SPLINE
SPL {X  -124.054, Y  +777.532, Z    +0.000, E1   -54.436, E3 +106436.833}
SPL {X  -145.922, Y  +742.101, Z    +0.000, E1   -46.535, E3 +106455.102}
SPL {X  -155.216, Y  +715.293, Z    +0.000, E1   -34.460, E3 +106461.295}
SPL {X  -158.715, Y  +696.660, Z    +0.000, E1   -21.368, E3 +106463.622}
SPL {X  -159.838, Y  +683.473, Z    +0.000, E1    -9.532, E3 +106464.418}
SPL {X  -159.990, Y  +674.579, Z    +0.000, E1    -0.168, E3 +106464.601}
SPL {X  -159.990, Y  +672.677, Z    +0.000, E1    +3.879, E3 +106464.617}
SPL {X  -159.990, Y  +669.117, Z    +0.000, E1   +12.900, E3 +106464.699}
SPL {X  -159.990, Y  +663.639, Z    +0.000, E1   +26.675, E3 +106464.985}
SPL {X  -159.990, Y  +656.057, Z    +0.000, E1   +43.288, E3 +106465.641}
SPL {X  -159.990, Y  +647.797, Z    +0.000, E1   +54.469, E3 +106466.778}
SPL {X  -159.990, Y  +630.178, Z    +0.000, E1   +65.480, E3 +106470.462}
SPL {X  -159.990, Y  +547.268, Z    +0.000, E1   +73.735, E3 +106497.746}
SPL {X  -159.091, Y  +360.560, Z    +0.000, E1   +74.726, E3 +106584.072}
SPL {X  -156.418, Y  +343.879, Z    +0.000, E1   +74.473, E3 +106596.498}
SPL {X  -153.414, Y  +332.103, Z    +0.000, E1   +74.378, E3 +106604.173}
SPL {X  -141.909, Y  +303.617, Z    +0.000, E1   +76.515, E3 +106596.703}
ENDSPLINE

SPLINE
SPL {X  -142.567, Y  +304.895, Z    +0.000, E1   +75.566, E3 +106605.518}
ENDSPLINE

SPLINE
SPL {X  -141.999, Y  +303.790, Z    +0.000, E1   +74.633, E3 +106614.769}
SPL {X  -141.780, Y  +303.371, Z    +0.000, E1   +73.549, E3 +106624.343}
SPL {X  -140.619, Y  +301.190, Z    +0.000, E1   +72.741, E3 +106632.189}
SPL {X  -137.438, Y  +295.601, Z    +0.000, E1   +72.365, E3 +106638.278}
SPL {X  -134.156, Y  +290.328, Z    +0.000, E1   +71.962, E3 +106644.149}
SPL {X  -130.677, Y  +285.194, Z    +0.000, E1   +71.519, E3 +106649.954}
SPL {X  -127.147, Y  +280.390, Z    +0.000, E1   +71.042, E3 +106655.438}
SPL {X  -123.431, Y  +275.709, Z    +0.000, E1   +70.518, E3 +106660.761}
SPL {X  -120.392, Y  +272.131, Z    +0.000, E1   +70.053, E3 +106664.781}
SPL {X   -79.311, Y  +238.552, Z    +0.000, E1   +58.563, E3 +106760.020}
ENDSPLINE

SPLINE
SPL {X  -105.077, Y  +256.854, Z    +0.000, E1   +55.187, E3 +106947.573}
SPL {X  -133.208, Y  +288.886, Z    +0.000, E1   +52.003, E3 +106980.674}
SPL {X  -149.825, Y  +321.381, Z    +0.000, E1   +42.580, E3 +106993.827}
SPL {X  -157.376, Y  +348.695, Z    +0.000, E1   +27.651, E3 +106998.912}
SPL {X  -159.486, Y  +364.808, Z    +0.000, E1   +14.693, E3 +107000.415}
SPL {X  -159.964, Y  +374.630, Z    +0.000, E1    +5.249, E3 +107000.820}
SPL {X  -159.990, Y  +379.735, Z    +0.000, E1    -0.236, E3 +107000.878}
SPL {X  -159.990, Y  +384.648, Z    +0.000, E1   -11.739, E3 +107000.974}
SPL {X  -159.990, Y  +391.065, Z    +0.000, E1   -28.187, E3 +107001.302}
SPL {X  -159.990, Y  +399.326, Z    +0.000, E1   -44.934, E3 +107002.085}
SPL {X  -159.990, Y  +408.817, Z    +0.000, E1   -56.572, E3 +107003.458}
SPL {X  -159.990, Y  +426.617, Z    +0.000, E1   -66.230, E3 +107007.313}
SPL {X  -159.990, Y  +499.521, Z    +0.000, E1   -73.662, E3 +107030.640}
SPL {X  -159.629, Y  +687.249, Z    +0.000, E1   -74.539, E3 +107118.524}
SPL {X  -157.983, Y  +701.765, Z    +0.000, E1   -74.384, E3 +107128.756}
SPL {X  -155.520, Y  +714.054, Z    +0.000, E1   -74.151, E3 +107138.510}
SPL {X  -152.569, Y  +724.660, Z    +0.000, E1   -73.857, E3 +107147.745}
SPL {X  -149.625, Y  +733.149, Z    +0.000, E1   -73.553, E3 +107155.680}
SPL {X  -146.617, Y  +740.532, Z    +0.000, E1   -73.233, E3 +107162.957}
SPL {X  -143.394, Y  +747.457, Z    +0.000, E1   -72.883, E3 +107170.054}
SPL {X  -140.332, Y  +753.336, Z    +0.000, E1   -72.527, E3 +107176.329}
SPL {X  -137.187, Y  +758.820, Z    +0.000, E1   -72.156, E3 +107182.332}
SPL {X  -134.014, Y  +763.891, Z    +0.000, E1   -71.759, E3 +107188.017}
SPL {X  -130.657, Y  +768.834, Z    +0.000, E1   -71.330, E3 +107193.632}
SPL {X  -126.937, Y  +773.885, Z    +0.000, E1   -70.823, E3 +107199.434}
SPL {X  -122.983, Y  +778.833, Z    +0.000, E1   -70.262, E3 +107205.079}
SPL {X  -120.205, Y  +782.082, Z    +0.000, E1   -69.822, E3 +107208.747}
SPL {X   -75.772, Y  +817.409, Z    +0.000, E1   -56.226, E3 +107334.686}
ENDSPLINE

SPLINE
SPL {X  -124.054, Y  +777.532, Z    +0.000, E1   -54.436, E3 +107517.914}
SPL {X  -145.922, Y  +742.101, Z    +0.000, E1   -46.535, E3 +107536.184}
SPL {X  -155.216, Y  +715.293, Z    +0.000, E1   -34.460, E3 +107542.376}
SPL {X  -159.282, Y  +691.530, Z    +0.000, E1   -17.100, E3 +107545.071}
SPL {X  -159.981, Y  +678.202, Z    +0.000, E1    -4.129, E3 +107545.645}
SPL {X  -159.990, Y  +674.500, Z    +0.000, E1    +0.000, E3 +107545.682}
SPL {X  -159.990, Y  +672.677, Z    +0.000, E1    +3.879, E3 +107545.698}
SPL {X  -159.990, Y  +669.117, Z    +0.000, E1   +12.900, E3 +107545.781}
SPL {X  -159.990, Y  +665.253, Z    +0.000, E1   +22.908, E3 +107545.954}
SPL {X  -159.990, Y  +658.335, Z    +0.000, E1   +38.839, E3 +107546.499}
SPL {X  -159.990, Y  +645.786, Z    +0.000, E1   +56.338, E3 +107548.213}
SPL {X  -159.990, Y  +623.264, Z    +0.000, E1   +67.753, E3 +107553.139}
SPL {X  -159.990, Y  +547.268, Z    +0.000, E1   +73.735, E3 +107578.827}
SPL {X  -159.091, Y  +360.560, Z    +0.000, E1   +74.726, E3 +107665.154}
SPL {X  -156.418, Y  +343.879, Z    +0.000, E1   +74.473, E3 +107677.579}
SPL {X  -153.414, Y  +332.103, Z    +0.000, E1   +74.378, E3 +107685.254}
SPL {X  -141.909, Y  +303.617, Z    +0.000, E1   +76.515, E3 +107677.784}
ENDSPLINE

SPLINE
SPL {X  -142.567, Y  +304.895, Z    +0.000, E1   +75.566, E3 +107686.599}
ENDSPLINE

SPLINE
SPL {X  -141.999, Y  +303.790, Z    +0.000, E1   +74.633, E3 +107695.850}
SPL {X  -141.780, Y  +303.371, Z    +0.000, E1   +73.549, E3 +107705.424}
ENDSPLINE

SPLINE
SPL {X  -146.767, Y  +313.812, Z    +0.000, E1   +70.623, E3 +107723.087}
ENDSPLINE

SPLINE
SPL {X  -143.180, Y  +306.112, Z    +0.000, E1   +70.169, E3 +107731.789}
SPL {X  -139.769, Y  +299.645, Z    +0.000, E1   +69.722, E3 +107739.355}
SPL {X  -136.083, Y  +293.369, Z    +0.000, E1   +69.227, E3 +107746.896}
SPL {X  -132.274, Y  +287.498, Z    +0.000, E1   +68.678, E3 +107754.116}
SPL {X  -128.237, Y  +281.834, Z    +0.000, E1   +68.080, E3 +107761.152}
SPL {X  -124.030, Y  +276.439, Z    +0.000, E1   +67.412, E3 +107767.870}
SPL {X   -89.505, Y  +244.889, Z    +0.000, E1   +58.168, E3 +107849.622}
ENDSPLINE

SPLINE
SPL {X  -111.763, Y  +263.019, Z    +0.000, E1   +52.505, E3 +108031.034}
SPL {X  -139.943, Y  +299.958, Z    +0.000, E1   +46.517, E3 +108065.374}
SPL {X  -154.122, Y  +334.569, Z    +0.000, E1   +33.405, E3 +108077.208}
SPL {X  -159.233, Y  +361.951, Z    +0.000, E1   +15.631, E3 +108081.387}
SPL {X  -159.983, Y  +375.952, Z    +0.000, E1    +3.555, E3 +108082.153}
SPL {X  -159.990, Y  +379.545, Z    +0.000, E1    -0.045, E3 +108082.200}
SPL {X  -159.990, Y  +382.058, Z    +0.000, E1    -4.728, E3 +108082.232}
SPL {X  -159.990, Y  +387.492, Z    +0.000, E1   -16.478, E3 +108082.457}
SPL {X  -159.990, Y  +395.172, Z    +0.000, E1   -33.361, E3 +108083.084}
SPL {X  -159.990, Y  +405.626, Z    +0.000, E1   -49.217, E3 +108084.608}
SPL {X  -159.990, Y  +423.679, Z    +0.000, E1   -61.834, E3 +108088.879}
SPL {X  -159.990, Y  +491.183, Z    +0.000, E1   -70.406, E3 +108115.268}
SPL {X  -159.990, Y  +644.105, Z    +0.000, E1   -71.828, E3 +108199.837}
SPL {X  -159.990, Y  +665.410, Z    +0.000, E1   -71.813, E3 +108214.734}
SPL {X  -159.784, Y  +684.619, Z    +0.000, E1   -71.795, E3 +108228.338}
SPL {X  -158.321, Y  +699.551, Z    +0.000, E1   -71.633, E3 +108240.290}
SPL {X  -155.878, Y  +712.540, Z    +0.000, E1   -71.376, E3 +108251.853}
SPL {X  -152.746, Y  +724.097, Z    +0.000, E1   -71.019, E3 +108263.104}
SPL {X  -149.840, Y  +732.578, Z    +0.000, E1   -70.669, E3 +108271.930}
SPL {X  -147.044, Y  +739.548, Z    +0.000, E1   -70.332, E3 +108279.524}
SPL {X  -143.437, Y  +747.371, Z    +0.000, E1   -69.890, E3 +108288.388}
SPL {X  -139.209, Y  +755.353, Z    +0.000, E1   -69.333, E3 +108297.815}
SPL {X  -135.354, Y  +761.800, Z    +0.000, E1   -68.789, E3 +108305.678}
SPL {X  -131.547, Y  +767.562, Z    +0.000, E1   -68.238, E3 +108312.847}
SPL {X  -127.113, Y  +773.655, Z    +0.000, E1   -67.565, E3 +108320.504}
SPL {X  -123.626, Y  +778.056, Z    +0.000, E1   -66.969, E3 +108326.064}
SPL {X   -86.110, Y  +811.340, Z    +0.000, E1   -55.142, E3 +108443.974}
ENDSPLINE

SPLINE
SPL {X  -126.688, Y  +774.208, Z    +0.000, E1   -50.278, E3 +108604.622}
SPL {X  -150.887, Y  +729.697, Z    +0.000, E1   -37.846, E3 +108628.478}
SPL {X  -158.568, Y  +697.780, Z    +0.000, E1   -19.721, E3 +108634.807}
SPL {X  -159.967, Y  +679.234, Z    +0.000, E1    -4.684, E3 +108636.142}
SPL {X  -159.990, Y  +674.465, Z    +0.000, E1    +0.035, E3 +108636.225}
SPL {X  -159.990, Y  +672.210, Z    +0.000, E1    +4.112, E3 +108636.252}
SPL {X  -159.990, Y  +668.446, Z    +0.000, E1   +12.084, E3 +108636.377}
SPL {X  -159.990, Y  +663.424, Z    +0.000, E1   +23.273, E3 +108636.703}
SPL {X  -159.990, Y  +655.288, Z    +0.000, E1   +39.016, E3 +108637.592}
SPL {X  -159.990, Y  +641.020, Z    +0.000, E1   +55.512, E3 +108640.131}
SPL {X  -159.990, Y  +618.237, Z    +0.000, E1   +65.205, E3 +108646.657}
SPL {X  -159.990, Y  +545.807, Z    +0.000, E1   +71.095, E3 +108675.710}
SPL {X  -149.334, Y  +320.087, Z    +0.000, E1   +77.218, E3 +108741.528}
SPL {X  -149.265, Y  +319.910, Z    +0.000, E1   +76.148, E3 +108753.642}
SPL {X  -149.092, Y  +319.462, Z    +0.000, E1   +75.437, E3 +108761.517}
ENDSPLINE

SPLINE
SPL {X  -149.679, Y  +320.993, Z    +0.000, E1   +74.493, E3 +108770.411}
SPL {X  -149.823, Y  +321.377, Z    +0.000, E1   +73.518, E3 +108779.768}
ENDSPLINE

SPLINE
SPL {X  -149.061, Y  +319.382, Z    +0.000, E1   +72.547, E3 +108790.010}
SPL {X  -148.201, Y  +317.223, Z    +0.000, E1   +71.184, E3 +108803.334}
SPL {X  -144.085, Y  +307.957, Z    +0.000, E1   +70.311, E3 +108816.581}
SPL {X  -139.769, Y  +299.645, Z    +0.000, E1   +69.722, E3 +108826.312}
SPL {X  -136.083, Y  +293.369, Z    +0.000, E1   +69.227, E3 +108833.853}
SPL {X  -132.274, Y  +287.498, Z    +0.000, E1   +68.678, E3 +108841.072}
SPL {X  -128.237, Y  +281.834, Z    +0.000, E1   +68.080, E3 +108848.109}
SPL {X  -124.030, Y  +276.439, Z    +0.000, E1   +67.412, E3 +108854.826}
SPL {X   -89.505, Y  +244.889, Z    +0.000, E1   +58.168, E3 +108936.578}
ENDSPLINE

SPLINE
SPL {X  -111.763, Y  +263.019, Z    +0.000, E1   +52.505, E3 +109117.990}
SPL {X  -139.943, Y  +299.958, Z    +0.000, E1   +46.517, E3 +109152.330}
SPL {X  -154.122, Y  +334.569, Z    +0.000, E1   +33.405, E3 +109164.165}
SPL {X  -159.233, Y  +361.951, Z    +0.000, E1   +15.631, E3 +109168.343}
SPL {X  -159.983, Y  +375.952, Z    +0.000, E1    +3.555, E3 +109169.110}
SPL {X  -159.990, Y  +379.545, Z    +0.000, E1    -0.045, E3 +109169.156}
SPL {X  -159.990, Y  +382.058, Z    +0.000, E1    -4.728, E3 +109169.188}
SPL {X  -159.990, Y  +385.965, Z    +0.000, E1   -13.291, E3 +109169.323}
SPL {X  -159.990, Y  +391.054, Z    +0.000, E1   -24.765, E3 +109169.655}
SPL {X  -159.990, Y  +400.233, Z    +0.000, E1   -42.011, E3 +109170.699}
SPL {X  -159.990, Y  +418.500, Z    +0.000, E1   -59.260, E3 +109174.544}
SPL {X  -159.990, Y  +491.183, Z    +0.000, E1   -70.406, E3 +109202.225}
SPL {X  -159.990, Y  +644.105, Z    +0.000, E1   -71.828, E3 +109286.793}
SPL {X  -159.990, Y  +665.410, Z    +0.000, E1   -71.813, E3 +109301.691}
SPL {X  -159.936, Y  +680.656, Z    +0.000, E1   -71.796, E3 +109312.408}
SPL {X  -158.712, Y  +696.685, Z    +0.000, E1   -71.696, E3 +109324.792}
SPL {X  -156.572, Y  +709.392, Z    +0.000, E1   -71.434, E3 +109335.939}
SPL {X  -154.409, Y  +718.389, Z    +0.000, E1   -71.209, E3 +109344.399}
SPL {X  -150.682, Y  +730.275, Z    +0.000, E1   -70.793, E3 +109356.398}
SPL {X  -147.044, Y  +739.548, Z    +0.000, E1   -70.332, E3 +109366.481}
SPL {X  -144.262, Y  +745.675, Z    +0.000, E1   -69.979, E3 +109373.419}
SPL {X  -141.227, Y  +751.679, Z    +0.000, E1   -69.593, E3 +109380.405}
SPL {X  -138.327, Y  +756.889, Z    +0.000, E1   -69.193, E3 +109386.655}
SPL {X  -134.311, Y  +763.433, Z    +0.000, E1   -68.667, E3 +109394.617}
SPL {X  -129.529, Y  +770.410, Z    +0.000, E1   -67.934, E3 +109403.381}
SPL {X  -126.163, Y  +774.886, Z    +0.000, E1   -67.384, E3 +109409.044}
SPL {X  -123.626, Y  +778.056, Z    +0.000, E1   -66.969, E3 +109413.021}
SPL {X   -86.110, Y  +811.340, Z    +0.000, E1   -55.142, E3 +109530.931}
ENDSPLINE

SPLINE
SPL {X  -126.688, Y  +774.208, Z    +0.000, E1   -50.278, E3 +109691.578}
SPL {X  -150.887, Y  +729.697, Z    +0.000, E1   -37.846, E3 +109715.434}
SPL {X  -157.603, Y  +704.031, Z    +0.000, E1   -23.939, E3 +109720.996}
SPL {X  -159.560, Y  +688.227, Z    +0.000, E1   -12.334, E3 +109722.670}
SPL {X  -159.987, Y  +677.470, Z    +0.000, E1    -2.943, E3 +109723.149}
SPL {X  -159.990, Y  +674.465, Z    +0.000, E1    +0.035, E3 +109723.181}
SPL {X  -159.990, Y  +672.210, Z    +0.000, E1    +4.112, E3 +109723.208}
SPL {X  -159.990, Y  +668.446, Z    +0.000, E1   +12.084, E3 +109723.334}
SPL {X  -159.990, Y  +663.424, Z    +0.000, E1   +23.273, E3 +109723.660}
SPL {X  -159.990, Y  +655.288, Z    +0.000, E1   +39.016, E3 +109724.549}
SPL {X  -159.990, Y  +641.020, Z    +0.000, E1   +55.512, E3 +109727.088}
SPL {X  -159.990, Y  +618.237, Z    +0.000, E1   +65.205, E3 +109733.613}
SPL {X  -159.990, Y  +545.807, Z    +0.000, E1   +71.095, E3 +109762.666}
SPL {X  -159.990, Y  +417.971, Z    +0.000, E1   +72.138, E3 +109831.326}
SPL {X  -147.674, Y  +315.943, Z    +0.000, E1   +77.803, E3 +109823.056}
ENDSPLINE

SPLINE
SPL {X  -149.193, Y  +319.722, Z    +0.000, E1   +76.912, E3 +109831.998}
ENDSPLINE

SPLINE
SPL {X  -149.153, Y  +319.620, Z    +0.000, E1   +75.840, E3 +109844.408}
ENDSPLINE

SPLINE
SPL {X  -149.679, Y  +320.993, Z    +0.000, E1   +74.493, E3 +109857.367}
SPL {X  -149.823, Y  +321.377, Z    +0.000, E1   +73.518, E3 +109866.725}
ENDSPLINE

SPLINE
SPL {X  -149.061, Y  +319.382, Z    +0.000, E1   +72.547, E3 +109876.966}
SPL {X  -148.522, Y  +318.020, Z    +0.000, E1   +71.446, E3 +109887.352}
SPL {X  -146.766, Y  +313.809, Z    +0.000, E1   +70.623, E3 +109897.004}
SPL {X  -143.180, Y  +306.112, Z    +0.000, E1   +70.169, E3 +109905.702}
SPL {X  -138.714, Y  +297.780, Z    +0.000, E1   +69.607, E3 +109915.448}
SPL {X  -135.202, Y  +291.959, Z    +0.000, E1   +69.085, E3 +109922.557}
SPL {X  -131.272, Y  +286.043, Z    +0.000, E1   +68.558, E3 +109929.796}
SPL {X  -127.436, Y  +280.769, Z    +0.000, E1   +67.934, E3 +109936.419}
SPL {X  -124.030, Y  +276.439, Z    +0.000, E1   +67.412, E3 +109941.783}
SPL {X   -89.505, Y  +244.889, Z    +0.000, E1   +58.168, E3 +110023.535}
ENDSPLINE

SPLINE
SPL {X  -111.763, Y  +263.019, Z    +0.000, E1   +52.505, E3 +110204.947}
SPL {X  -139.943, Y  +299.958, Z    +0.000, E1   +46.517, E3 +110239.287}
SPL {X  -152.249, Y  +328.336, Z    +0.000, E1   +36.404, E3 +110249.681}
SPL {X  -158.157, Y  +353.354, Z    +0.000, E1   +21.990, E3 +110254.405}
SPL {X  -159.828, Y  +370.311, Z    +0.000, E1    +8.652, E3 +110255.870}
SPL {X  -159.990, Y  +377.723, Z    +0.000, E1    +1.782, E3 +110256.101}
SPL {X  -159.990, Y  +379.545, Z    +0.000, E1    -0.045, E3 +110256.113}
SPL {X  -159.990, Y  +382.058, Z    +0.000, E1    -4.728, E3 +110256.145}
SPL {X  -159.990, Y  +387.492, Z    +0.000, E1   -16.478, E3 +110256.370}
SPL {X  -159.990, Y  +395.172, Z    +0.000, E1   -33.361, E3 +110256.997}
SPL {X  -159.990, Y  +405.626, Z    +0.000, E1   -49.217, E3 +110258.521}
SPL {X  -159.990, Y  +423.679, Z    +0.000, E1   -61.834, E3 +110262.792}
SPL {X  -159.990, Y  +491.183, Z    +0.000, E1   -70.406, E3 +110289.181}
SPL {X  -159.990, Y  +644.105, Z    +0.000, E1   -71.828, E3 +110373.750}
SPL {X  -159.990, Y  +665.410, Z    +0.000, E1   -71.813, E3 +110388.647}
SPL {X  -159.784, Y  +684.619, Z    +0.000, E1   -71.795, E3 +110402.251}
SPL {X  -158.321, Y  +699.551, Z    +0.000, E1   -71.633, E3 +110414.203}
SPL {X  -155.878, Y  +712.540, Z    +0.000, E1   -71.376, E3 +110425.766}
SPL {X  -152.746, Y  +724.097, Z    +0.000, E1   -71.019, E3 +110437.017}
SPL {X  -149.840, Y  +732.578, Z    +0.000, E1   -70.669, E3 +110445.843}
SPL {X  -147.044, Y  +739.548, Z    +0.000, E1   -70.332, E3 +110453.437}
SPL {X  -144.262, Y  +745.675, Z    +0.000, E1   -69.979, E3 +110460.375}
SPL {X  -141.227, Y  +751.679, Z    +0.000, E1   -69.593, E3 +110467.361}
SPL {X  -138.327, Y  +756.889, Z    +0.000, E1   -69.193, E3 +110473.612}
SPL {X  -135.354, Y  +761.800, Z    +0.000, E1   -68.789, E3 +110479.591}
SPL {X  -131.547, Y  +767.562, Z    +0.000, E1   -68.238, E3 +110486.760}
SPL {X  -128.543, Y  +771.755, Z    +0.000, E1   -67.757, E3 +110492.061}
SPL {X  -126.163, Y  +774.886, Z    +0.000, E1   -67.384, E3 +110496.000}
SPL {X  -123.626, Y  +778.056, Z    +0.000, E1   -66.969, E3 +110499.977}
SPL {X   -86.110, Y  +811.340, Z    +0.000, E1   -55.142, E3 +110617.887}
ENDSPLINE

SPLINE
SPL {X  -126.688, Y  +774.208, Z    +0.000, E1   -50.278, E3 +110778.535}
SPL {X  -150.887, Y  +729.697, Z    +0.000, E1   -37.846, E3 +110802.391}
SPL {X  -158.568, Y  +697.780, Z    +0.000, E1   -19.721, E3 +110808.720}
SPL {X  -159.967, Y  +679.234, Z    +0.000, E1    -4.684, E3 +110810.055}
SPL {X  -159.990, Y  +674.465, Z    +0.000, E1    +0.035, E3 +110810.138}
SPL {X  -159.990, Y  +672.210, Z    +0.000, E1    +4.112, E3 +110810.165}
SPL {X  -159.990, Y  +668.446, Z    +0.000, E1   +12.084, E3 +110810.290}
SPL {X  -159.990, Y  +663.424, Z    +0.000, E1   +23.273, E3 +110810.616}
SPL {X  -159.990, Y  +655.288, Z    +0.000, E1   +39.016, E3 +110811.505}
SPL {X  -159.990, Y  +641.020, Z    +0.000, E1   +55.512, E3 +110814.044}
SPL {X  -159.990, Y  +618.237, Z    +0.000, E1   +65.205, E3 +110820.570}
SPL {X  -159.990, Y  +545.807, Z    +0.000, E1   +71.095, E3 +110849.623}
SPL {X  -159.990, Y  +417.971, Z    +0.000, E1   +72.138, E3 +110918.282}
SPL {X  -147.674, Y  +315.943, Z    +0.000, E1   +77.803, E3 +110910.013}
ENDSPLINE

SPLINE
SPL {X  -149.193, Y  +319.722, Z    +0.000, E1   +76.912, E3 +110918.955}
ENDSPLINE

SPLINE
SPL {X  -149.153, Y  +319.620, Z    +0.000, E1   +75.840, E3 +110931.364}
ENDSPLINE

SPLINE
SPL {X  -149.679, Y  +320.993, Z    +0.000, E1   +74.493, E3 +110944.324}
SPL {X  -149.823, Y  +321.377, Z    +0.000, E1   +73.518, E3 +110953.681}
ENDSPLINE

SPLINE
SPL {X  -149.061, Y  +319.382, Z    +0.000, E1   +72.547, E3 +110963.923}
SPL {X  -148.201, Y  +317.223, Z    +0.000, E1   +71.184, E3 +110977.247}
SPL {X  -144.085, Y  +307.957, Z    +0.000, E1   +70.311, E3 +110990.494}
SPL {X  -139.769, Y  +299.645, Z    +0.000, E1   +69.722, E3 +111000.225}
SPL {X  -136.083, Y  +293.369, Z    +0.000, E1   +69.227, E3 +111007.766}
SPL {X  -131.272, Y  +286.043, Z    +0.000, E1   +68.558, E3 +111016.752}
SPL {X  -127.436, Y  +280.769, Z    +0.000, E1   +67.934, E3 +111023.376}
SPL {X  -124.030, Y  +276.439, Z    +0.000, E1   +67.412, E3 +111028.739}
SPL {X   -89.505, Y  +244.889, Z    +0.000, E1   +58.168, E3 +111110.491}
ENDSPLINE

SPLINE
SPL {X  -111.763, Y  +263.019, Z    +0.000, E1   +52.505, E3 +111291.903}
SPL {X  -139.943, Y  +299.958, Z    +0.000, E1   +46.517, E3 +111326.243}
SPL {X  -152.249, Y  +328.336, Z    +0.000, E1   +36.404, E3 +111336.638}
SPL {X  -158.157, Y  +353.354, Z    +0.000, E1   +21.990, E3 +111341.361}
SPL {X  -159.630, Y  +366.769, Z    +0.000, E1   +11.595, E3 +111342.643}
SPL {X  -159.983, Y  +375.952, Z    +0.000, E1    +3.555, E3 +111343.023}
SPL {X  -159.990, Y  +379.545, Z    +0.000, E1    -0.045, E3 +111343.069}
SPL {X  -159.990, Y  +382.058, Z    +0.000, E1    -4.728, E3 +111343.101}
SPL {X  -159.990, Y  +387.492, Z    +0.000, E1   -16.478, E3 +111343.327}
SPL {X  -159.990, Y  +395.172, Z    +0.000, E1   -33.361, E3 +111343.954}
SPL {X  -159.990, Y  +405.626, Z    +0.000, E1   -49.217, E3 +111345.477}
SPL {X  -159.990, Y  +423.679, Z    +0.000, E1   -61.834, E3 +111349.749}
SPL {X  -159.990, Y  +491.183, Z    +0.000, E1   -70.406, E3 +111376.138}
SPL {X  -159.990, Y  +644.105, Z    +0.000, E1   -71.828, E3 +111460.706}
SPL {X  -159.990, Y  +665.410, Z    +0.000, E1   -71.813, E3 +111475.604}
SPL {X  -159.784, Y  +684.619, Z    +0.000, E1   -71.795, E3 +111489.207}
SPL {X  -158.321, Y  +699.551, Z    +0.000, E1   -71.633, E3 +111501.159}
SPL {X  -155.878, Y  +712.540, Z    +0.000, E1   -71.376, E3 +111512.723}
SPL {X  -152.746, Y  +724.097, Z    +0.000, E1   -71.019, E3 +111523.974}
SPL {X  -149.840, Y  +732.578, Z    +0.000, E1   -70.669, E3 +111532.800}
SPL {X  -147.044, Y  +739.548, Z    +0.000, E1   -70.332, E3 +111540.394}
SPL {X  -143.437, Y  +747.371, Z    +0.000, E1   -69.890, E3 +111549.257}
SPL {X  -139.209, Y  +755.353, Z    +0.000, E1   -69.333, E3 +111558.684}
SPL {X  -135.354, Y  +761.800, Z    +0.000, E1   -68.789, E3 +111566.548}
SPL {X  -131.547, Y  +767.562, Z    +0.000, E1   -68.238, E3 +111573.717}
SPL {X  -127.113, Y  +773.655, Z    +0.000, E1   -67.565, E3 +111581.373}
SPL {X  -123.626, Y  +778.056, Z    +0.000, E1   -66.969, E3 +111586.934}
SPL {X   -86.110, Y  +811.340, Z    +0.000, E1   -55.142, E3 +111704.844}
ENDSPLINE

SPLINE
SPL {X  -126.688, Y  +774.208, Z    +0.000, E1   -50.278, E3 +111865.491}
SPL {X  -147.153, Y  +739.291, Z    +0.000, E1   -41.559, E3 +111886.326}
SPL {X  -156.578, Y  +709.366, Z    +0.000, E1   -27.394, E3 +111894.018}
SPL {X  -159.560, Y  +688.227, Z    +0.000, E1   -12.334, E3 +111896.583}
SPL {X  -159.987, Y  +677.470, Z    +0.000, E1    -2.943, E3 +111897.062}
SPL {X  -159.990, Y  +674.465, Z    +0.000, E1    +0.035, E3 +111897.094}
SPL {X  -159.990, Y  +672.210, Z    +0.000, E1    +4.112, E3 +111897.121}
SPL {X  -159.990, Y  +668.446, Z    +0.000, E1   +12.084, E3 +111897.247}
SPL {X  -159.990, Y  +663.424, Z    +0.000, E1   +23.273, E3 +111897.573}
SPL {X  -159.990, Y  +655.288, Z    +0.000, E1   +39.016, E3 +111898.462}
SPL {X  -159.990, Y  +641.020, Z    +0.000, E1   +55.512, E3 +111901.001}
SPL {X  -159.990, Y  +618.237, Z    +0.000, E1   +65.205, E3 +111907.526}
SPL {X  -159.990, Y  +545.807, Z    +0.000, E1   +71.095, E3 +111936.579}
SPL {X  -159.990, Y  +417.971, Z    +0.000, E1   +72.138, E3 +112005.239}
SPL {X  -147.674, Y  +315.943, Z    +0.000, E1   +77.803, E3 +111996.970}
ENDSPLINE

SPLINE
SPL {X  -149.193, Y  +319.722, Z    +0.000, E1   +76.912, E3 +112005.911}
ENDSPLINE

SPLINE
SPL {X  -149.153, Y  +319.620, Z    +0.000, E1   +75.840, E3 +112018.321}
ENDSPLINE

SPLINE
SPL {X  -149.679, Y  +320.993, Z    +0.000, E1   +74.493, E3 +112031.280}
SPL {X  -149.823, Y  +321.377, Z    +0.000, E1   +73.518, E3 +112040.638}
ENDSPLINE

SPLINE
SPL {X  -149.061, Y  +319.382, Z    +0.000, E1   +72.547, E3 +112050.879}
SPL {X  -148.522, Y  +318.020, Z    +0.000, E1   +71.446, E3 +112061.265}
SPL {X  -146.766, Y  +313.809, Z    +0.000, E1   +70.623, E3 +112070.917}
SPL {X  -143.180, Y  +306.112, Z    +0.000, E1   +70.169, E3 +112079.615}
SPL {X  -139.769, Y  +299.645, Z    +0.000, E1   +69.722, E3 +112087.181}
SPL {X  -136.083, Y  +293.369, Z    +0.000, E1   +69.227, E3 +112094.722}
SPL {X  -132.274, Y  +287.498, Z    +0.000, E1   +68.678, E3 +112101.942}
SPL {X  -128.237, Y  +281.834, Z    +0.000, E1   +68.080, E3 +112108.978}
SPL {X  -125.186, Y  +277.874, Z    +0.000, E1   +67.573, E3 +112113.945}
SPL {X  -123.070, Y  +275.272, Z    +0.000, E1   +67.229, E3 +112117.165}
SPL {X   -89.505, Y  +244.889, Z    +0.000, E1   +58.168, E3 +112197.448}
ENDSPLINE

SPLINE
SPL {X  -111.763, Y  +263.019, Z    +0.000, E1   +52.505, E3 +112378.860}
SPL {X  -139.943, Y  +299.958, Z    +0.000, E1   +46.517, E3 +112413.200}
SPL {X  -154.122, Y  +334.569, Z    +0.000, E1   +33.405, E3 +112425.034}
SPL {X  -159.233, Y  +361.951, Z    +0.000, E1   +15.631, E3 +112429.213}
SPL {X  -159.983, Y  +375.952, Z    +0.000, E1    +3.555, E3 +112429.980}
SPL {X  -159.990, Y  +379.545, Z    +0.000, E1    -0.045, E3 +112430.026}
SPL {X  -159.990, Y  +382.058, Z    +0.000, E1    -4.728, E3 +112430.058}
SPL {X  -159.990, Y  +385.965, Z    +0.000, E1   -13.291, E3 +112430.192}
SPL {X  -159.990, Y  +391.054, Z    +0.000, E1   -24.765, E3 +112430.524}
SPL {X  -159.990, Y  +400.233, Z    +0.000, E1   -42.011, E3 +112431.569}
SPL {X  -159.990, Y  +418.500, Z    +0.000, E1   -59.260, E3 +112435.413}
SPL {X  -159.990, Y  +491.183, Z    +0.000, E1   -70.406, E3 +112463.094}
SPL {X  -159.990, Y  +644.105, Z    +0.000, E1   -71.828, E3 +112547.663}
SPL {X  -159.990, Y  +665.410, Z    +0.000, E1   -71.813, E3 +112562.560}
SPL {X  -159.784, Y  +684.619, Z    +0.000, E1   -71.795, E3 +112576.164}
SPL {X  -158.321, Y  +699.551, Z    +0.000, E1   -71.633, E3 +112588.116}
SPL {X  -155.878, Y  +712.540, Z    +0.000, E1   -71.376, E3 +112599.679}
SPL {X  -152.746, Y  +724.097, Z    +0.000, E1   -71.019, E3 +112610.930}
SPL {X  -149.840, Y  +732.578, Z    +0.000, E1   -70.669, E3 +112619.756}
SPL {X  -147.044, Y  +739.548, Z    +0.000, E1   -70.332, E3 +112627.350}
SPL {X  -143.437, Y  +747.371, Z    +0.000, E1   -69.890, E3 +112636.214}
SPL {X  -139.209, Y  +755.353, Z    +0.000, E1   -69.333, E3 +112645.641}
SPL {X  -135.354, Y  +761.800, Z    +0.000, E1   -68.789, E3 +112653.504}
SPL {X  -131.547, Y  +767.562, Z    +0.000, E1   -68.238, E3 +112660.673}
SPL {X  -128.543, Y  +771.755, Z    +0.000, E1   -67.757, E3 +112665.974}
SPL {X  -126.163, Y  +774.886, Z    +0.000, E1   -67.384, E3 +112669.913}
SPL {X  -123.626, Y  +778.056, Z    +0.000, E1   -66.969, E3 +112673.890}
SPL {X   -86.110, Y  +811.340, Z    +0.000, E1   -55.142, E3 +112791.800}
ENDSPLINE

SPLINE
SPL {X  -126.688, Y  +774.208, Z    +0.000, E1   -50.278, E3 +112952.448}
SPL {X  -147.153, Y  +739.291, Z    +0.000, E1   -41.559, E3 +112973.282}
SPL {X  -156.578, Y  +709.366, Z    +0.000, E1   -27.394, E3 +112980.975}
SPL {X  -159.560, Y  +688.227, Z    +0.000, E1   -12.334, E3 +112983.540}
SPL {X  -159.987, Y  +677.470, Z    +0.000, E1    -2.943, E3 +112984.019}
SPL {X  -159.990, Y  +674.465, Z    +0.000, E1    +0.035, E3 +112984.051}
SPL {X  -159.990, Y  +672.210, Z    +0.000, E1    +4.112, E3 +112984.078}
SPL {X  -159.990, Y  +668.446, Z    +0.000, E1   +12.084, E3 +112984.203}
SPL {X  -159.990, Y  +663.424, Z    +0.000, E1   +23.273, E3 +112984.529}
SPL {X  -159.990, Y  +655.288, Z    +0.000, E1   +39.016, E3 +112985.418}
SPL {X  -159.990, Y  +641.020, Z    +0.000, E1   +55.512, E3 +112987.957}
SPL {X  -159.990, Y  +618.237, Z    +0.000, E1   +65.205, E3 +112994.483}
SPL {X  -159.990, Y  +545.807, Z    +0.000, E1   +71.095, E3 +113023.536}
SPL {X  -159.990, Y  +417.971, Z    +0.000, E1   +72.138, E3 +113092.195}
SPL {X  -147.674, Y  +315.943, Z    +0.000, E1   +77.803, E3 +113083.926}
ENDSPLINE

SPLINE
SPL {X  -149.193, Y  +319.722, Z    +0.000, E1   +76.912, E3 +113092.868}
ENDSPLINE

SPLINE
SPL {X  -149.153, Y  +319.620, Z    +0.000, E1   +75.840, E3 +113105.277}
ENDSPLINE

SPLINE
SPL {X  -149.679, Y  +320.993, Z    +0.000, E1   +74.493, E3 +113118.237}
SPL {X  -149.823, Y  +321.377, Z    +0.000, E1   +73.518, E3 +113127.594}
ENDSPLINE

SPLINE
SPL {X  -149.061, Y  +319.382, Z    +0.000, E1   +72.547, E3 +113137.836}
SPL {X  -148.201, Y  +317.223, Z    +0.000, E1   +71.184, E3 +113151.161}
SPL {X  -144.085, Y  +307.957, Z    +0.000, E1   +70.311, E3 +113164.407}
SPL {X  -138.714, Y  +297.780, Z    +0.000, E1   +69.607, E3 +113176.317}
SPL {X  -135.202, Y  +291.959, Z    +0.000, E1   +69.085, E3 +113183.426}
SPL {X  -132.274, Y  +287.498, Z    +0.000, E1   +68.678, E3 +113188.898}
SPL {X  -128.237, Y  +281.834, Z    +0.000, E1   +68.080, E3 +113195.935}
SPL {X  -125.186, Y  +277.874, Z    +0.000, E1   +67.573, E3 +113200.902}
SPL {X  -123.070, Y  +275.272, Z    +0.000, E1   +67.229, E3 +113204.121}
SPL {X   -89.505, Y  +244.889, Z    +0.000, E1   +58.168, E3 +113284.404}
ENDSPLINE

SPLINE
SPL {X  -111.763, Y  +263.019, Z    +0.000, E1   +52.505, E3 +113465.816}
SPL {X  -139.943, Y  +299.958, Z    +0.000, E1   +46.517, E3 +113500.157}
SPL {X  -152.249, Y  +328.336, Z    +0.000, E1   +36.404, E3 +113510.551}
SPL {X  -158.157, Y  +353.354, Z    +0.000, E1   +21.990, E3 +113515.274}
SPL {X  -159.630, Y  +366.769, Z    +0.000, E1   +11.595, E3 +113516.556}
SPL {X  -159.983, Y  +375.952, Z    +0.000, E1    +3.555, E3 +113516.936}
SPL {X  -159.990, Y  +379.545, Z    +0.000, E1    -0.045, E3 +113516.982}
SPL {X  -159.990, Y  +382.058, Z    +0.000, E1    -4.728, E3 +113517.015}
SPL {X  -159.990, Y  +387.492, Z    +0.000, E1   -16.478, E3 +113517.240}
SPL {X  -159.990, Y  +395.172, Z    +0.000, E1   -33.361, E3 +113517.867}
SPL {X  -159.990, Y  +405.626, Z    +0.000, E1   -49.217, E3 +113519.390}
SPL {X  -159.990, Y  +423.679, Z    +0.000, E1   -61.834, E3 +113523.662}
SPL {X  -159.990, Y  +491.183, Z    +0.000, E1   -70.406, E3 +113550.051}
SPL {X  -159.990, Y  +644.105, Z    +0.000, E1   -71.828, E3 +113634.619}
SPL {X  -159.990, Y  +665.410, Z    +0.000, E1   -71.813, E3 +113649.517}
SPL {X  -159.784, Y  +684.619, Z    +0.000, E1   -71.795, E3 +113663.120}
SPL {X  -158.321, Y  +699.551, Z    +0.000, E1   -71.633, E3 +113675.072}
SPL {X  -155.878, Y  +712.540, Z    +0.000, E1   -71.376, E3 +113686.636}
SPL {X  -152.746, Y  +724.097, Z    +0.000, E1   -71.019, E3 +113697.887}
SPL {X  -149.840, Y  +732.578, Z    +0.000, E1   -70.669, E3 +113706.713}
SPL {X  -147.044, Y  +739.548, Z    +0.000, E1   -70.332, E3 +113714.307}
SPL {X  -143.437, Y  +747.371, Z    +0.000, E1   -69.890, E3 +113723.170}
SPL {X  -139.209, Y  +755.353, Z    +0.000, E1   -69.333, E3 +113732.597}
SPL {X  -134.311, Y  +763.433, Z    +0.000, E1   -68.667, E3 +113742.443}
SPL {X  -129.529, Y  +770.410, Z    +0.000, E1   -67.934, E3 +113751.207}
SPL {X  -126.163, Y  +774.886, Z    +0.000, E1   -67.384, E3 +113756.870}
SPL {X  -123.626, Y  +778.056, Z    +0.000, E1   -66.969, E3 +113760.847}
SPL {X   -86.110, Y  +811.340, Z    +0.000, E1   -55.142, E3 +113878.757}
ENDSPLINE

SPLINE
SPL {X  -126.688, Y  +774.208, Z    +0.000, E1   -50.278, E3 +114039.404}
SPL {X  -150.887, Y  +729.697, Z    +0.000, E1   -37.846, E3 +114063.260}
SPL {X  -158.568, Y  +697.780, Z    +0.000, E1   -19.721, E3 +114069.590}
SPL {X  -159.967, Y  +679.234, Z    +0.000, E1    -4.684, E3 +114070.925}
SPL {X  -159.990, Y  +674.465, Z    +0.000, E1    +0.035, E3 +114071.008}
SPL {X  -159.990, Y  +672.210, Z    +0.000, E1    +4.112, E3 +114071.034}
SPL {X  -159.990, Y  +668.446, Z    +0.000, E1   +12.084, E3 +114071.160}
SPL {X  -159.990, Y  +663.424, Z    +0.000, E1   +23.273, E3 +114071.486}
SPL {X  -159.990, Y  +655.288, Z    +0.000, E1   +39.016, E3 +114072.375}
SPL {X  -159.990, Y  +641.020, Z    +0.000, E1   +55.512, E3 +114074.914}
SPL {X  -159.990, Y  +618.237, Z    +0.000, E1   +65.205, E3 +114081.439}
SPL {X  -159.990, Y  +545.807, Z    +0.000, E1   +71.095, E3 +114110.492}
SPL {X  -159.990, Y  +417.971, Z    +0.000, E1   +72.138, E3 +114179.152}
SPL {X  -147.674, Y  +315.943, Z    +0.000, E1   +77.803, E3 +114170.883}
ENDSPLINE

SPLINE
SPL {X  -149.193, Y  +319.722, Z    +0.000, E1   +76.912, E3 +114179.824}
ENDSPLINE

SPLINE
SPL {X  -149.153, Y  +319.620, Z    +0.000, E1   +75.840, E3 +114192.234}
ENDSPLINE

SPLINE
SPL {X  -149.679, Y  +320.993, Z    +0.000, E1   +74.493, E3 +114205.193}
SPL {X  -149.823, Y  +321.377, Z    +0.000, E1   +73.518, E3 +114214.551}
ENDSPLINE

SPLINE
SPL {X  -149.061, Y  +319.382, Z    +0.000, E1   +72.547, E3 +114224.792}
SPL {X  -148.201, Y  +317.223, Z    +0.000, E1   +71.184, E3 +114238.117}
SPL {X  -144.085, Y  +307.957, Z    +0.000, E1   +70.311, E3 +114251.364}
SPL {X  -139.769, Y  +299.645, Z    +0.000, E1   +69.722, E3 +114261.094}
SPL {X  -136.083, Y  +293.369, Z    +0.000, E1   +69.227, E3 +114268.636}
SPL {X  -131.272, Y  +286.043, Z    +0.000, E1   +68.558, E3 +114277.622}
SPL {X  -127.436, Y  +280.769, Z    +0.000, E1   +67.934, E3 +114284.245}
SPL {X  -124.030, Y  +276.439, Z    +0.000, E1   +67.412, E3 +114289.609}
SPL {X   -89.505, Y  +244.889, Z    +0.000, E1   +58.168, E3 +114371.361}
ENDSPLINE

SPLINE
SPL {X  -111.763, Y  +263.019, Z    +0.000, E1   +52.505, E3 +114552.773}
SPL {X  -139.943, Y  +299.958, Z    +0.000, E1   +46.517, E3 +114587.113}
SPL {X  -152.249, Y  +328.336, Z    +0.000, E1   +36.404, E3 +114597.507}
SPL {X  -158.157, Y  +353.354, Z    +0.000, E1   +21.990, E3 +114602.231}
SPL {X  -159.828, Y  +370.311, Z    +0.000, E1    +8.652, E3 +114603.696}
SPL {X  -159.990, Y  +377.723, Z    +0.000, E1    +1.782, E3 +114603.927}
SPL {X  -159.990, Y  +379.545, Z    +0.000, E1    -0.045, E3 +114603.939}
SPL {X  -159.990, Y  +382.058, Z    +0.000, E1    -4.728, E3 +114603.971}
SPL {X  -159.990, Y  +387.492, Z    +0.000, E1   -16.478, E3 +114604.196}
SPL {X  -159.990, Y  +395.172, Z    +0.000, E1   -33.361, E3 +114604.823}
SPL {X  -159.990, Y  +403.640, Z    +0.000, E1   -46.960, E3 +114605.971}
SPL {X  -159.990, Y  +418.500, Z    +0.000, E1   -59.260, E3 +114609.326}
SPL {X  -159.990, Y  +491.183, Z    +0.000, E1   -70.406, E3 +114637.007}
SPL {X  -159.990, Y  +636.738, Z    +0.000, E1   -71.802, E3 +114716.505}
SPL {X  -159.990, Y  +649.462, Z    +0.000, E1   -71.804, E3 +114725.374}
SPL {X  -159.990, Y  +665.410, Z    +0.000, E1   -71.813, E3 +114736.473}
SPL {X  -159.784, Y  +684.619, Z    +0.000, E1   -71.795, E3 +114750.077}
SPL {X  -158.321, Y  +699.551, Z    +0.000, E1   -71.633, E3 +114762.029}
SPL {X  -155.878, Y  +712.540, Z    +0.000, E1   -71.376, E3 +114773.592}
SPL {X  -152.746, Y  +724.097, Z    +0.000, E1   -71.019, E3 +114784.843}
SPL {X  -149.840, Y  +732.578, Z    +0.000, E1   -70.669, E3 +114793.669}
SPL {X  -147.044, Y  +739.548, Z    +0.000, E1   -70.332, E3 +114801.263}
SPL {X  -144.262, Y  +745.675, Z    +0.000, E1   -69.979, E3 +114808.201}
SPL {X  -141.227, Y  +751.679, Z    +0.000, E1   -69.593, E3 +114815.188}
SPL {X  -138.327, Y  +756.889, Z    +0.000, E1   -69.193, E3 +114821.438}
SPL {X  -135.354, Y  +761.800, Z    +0.000, E1   -68.789, E3 +114827.417}
SPL {X  -131.547, Y  +767.562, Z    +0.000, E1   -68.238, E3 +114834.586}
SPL {X  -128.543, Y  +771.755, Z    +0.000, E1   -67.757, E3 +114839.887}
SPL {X  -126.163, Y  +774.886, Z    +0.000, E1   -67.384, E3 +114843.826}
SPL {X  -123.626, Y  +778.056, Z    +0.000, E1   -66.969, E3 +114847.803}
SPL {X   -86.110, Y  +811.340, Z    +0.000, E1   -55.142, E3 +114965.714}
ENDSPLINE

SPLINE
SPL {X  -126.688, Y  +774.208, Z    +0.000, E1   -50.278, E3 +115126.361}
SPL {X  -150.887, Y  +729.697, Z    +0.000, E1   -37.846, E3 +115150.217}
SPL {X  -158.568, Y  +697.780, Z    +0.000, E1   -19.721, E3 +115156.546}
SPL {X  -159.967, Y  +679.234, Z    +0.000, E1    -4.684, E3 +115157.881}
SPL {X  -159.990, Y  +674.465, Z    +0.000, E1    +0.035, E3 +115157.964}
SPL {X  -159.990, Y  +672.210, Z    +0.000, E1    +4.112, E3 +115157.991}
SPL {X  -159.990, Y  +668.446, Z    +0.000, E1   +12.084, E3 +115158.116}
SPL {X  -159.990, Y  +663.424, Z    +0.000, E1   +23.273, E3 +115158.443}
SPL {X  -159.990, Y  +655.288, Z    +0.000, E1   +39.016, E3 +115159.331}
SPL {X  -159.990, Y  +641.020, Z    +0.000, E1   +55.512, E3 +115161.871}
SPL {X  -159.990, Y  +618.237, Z    +0.000, E1   +65.205, E3 +115168.396}
SPL {X  -159.990, Y  +545.807, Z    +0.000, E1   +71.095, E3 +115197.449}
SPL {X  -149.334, Y  +320.087, Z    +0.000, E1   +77.218, E3 +115263.267}
SPL {X  -149.265, Y  +319.910, Z    +0.000, E1   +76.148, E3 +115275.381}
SPL {X  -149.092, Y  +319.462, Z    +0.000, E1   +75.437, E3 +115283.256}
ENDSPLINE

SPLINE
SPL {X  -149.679, Y  +320.993, Z    +0.000, E1   +74.493, E3 +115292.150}
SPL {X  -149.823, Y  +321.377, Z    +0.000, E1   +73.518, E3 +115301.507}
ENDSPLINE

SPLINE
SPL {X  -149.061, Y  +319.382, Z    +0.000, E1   +72.547, E3 +115311.749}
SPL {X  -148.201, Y  +317.223, Z    +0.000, E1   +71.184, E3 +115325.074}
SPL {X  -144.085, Y  +307.957, Z    +0.000, E1   +70.311, E3 +115338.320}
SPL {X  -139.769, Y  +299.645, Z    +0.000, E1   +69.722, E3 +115348.051}
SPL {X  -136.083, Y  +293.369, Z    +0.000, E1   +69.227, E3 +115355.592}
SPL {X  -132.274, Y  +287.498, Z    +0.000, E1   +68.678, E3 +115362.811}
SPL {X  -128.237, Y  +281.834, Z    +0.000, E1   +68.080, E3 +115369.848}
SPL {X  -124.030, Y  +276.439, Z    +0.000, E1   +67.412, E3 +115376.565}
SPL {X   -89.505, Y  +244.889, Z    +0.000, E1   +58.168, E3 +115458.317}
ENDSPLINE

SPLINE
SPL {X  -111.763, Y  +263.019, Z    +0.000, E1   +52.505, E3 +115639.729}
SPL {X  -139.943, Y  +299.958, Z    +0.000, E1   +46.517, E3 +115674.070}
SPL {X  -154.122, Y  +334.569, Z    +0.000, E1   +33.405, E3 +115685.904}
SPL {X  -159.233, Y  +361.951, Z    +0.000, E1   +15.631, E3 +115690.082}
SPL {X  -159.983, Y  +375.952, Z    +0.000, E1    +3.555, E3 +115690.849}
SPL {X  -159.990, Y  +379.545, Z    +0.000, E1    -0.045, E3 +115690.896}
SPL {X  -159.990, Y  +382.058, Z    +0.000, E1    -4.728, E3 +115690.928}
SPL {X  -159.990, Y  +385.965, Z    +0.000, E1   -13.291, E3 +115691.062}
SPL {X  -159.990, Y  +391.054, Z    +0.000, E1   -24.765, E3 +115691.394}
SPL {X  -159.990, Y  +400.233, Z    +0.000, E1   -42.011, E3 +115692.438}
SPL {X  -159.990, Y  +418.500, Z    +0.000, E1   -59.260, E3 +115696.283}
SPL {X  -159.990, Y  +491.183, Z    +0.000, E1   -70.406, E3 +115723.964}
SPL {X  -159.990, Y  +644.105, Z    +0.000, E1   -71.828, E3 +115808.532}
SPL {X  -159.990, Y  +665.410, Z    +0.000, E1   -71.813, E3 +115823.430}
SPL {X  -159.784, Y  +684.619, Z    +0.000, E1   -71.795, E3 +115837.033}
SPL {X  -158.321, Y  +699.551, Z    +0.000, E1   -71.633, E3 +115848.986}
SPL {X  -155.878, Y  +712.540, Z    +0.000, E1   -71.376, E3 +115860.549}
SPL {X  -152.746, Y  +724.097, Z    +0.000, E1   -71.019, E3 +115871.800}
SPL {X  -149.840, Y  +732.578, Z    +0.000, E1   -70.669, E3 +115880.626}
SPL {X  -147.044, Y  +739.548, Z    +0.000, E1   -70.332, E3 +115888.220}
SPL {X  -143.437, Y  +747.371, Z    +0.000, E1   -69.890, E3 +115897.083}
SPL {X  -139.209, Y  +755.353, Z    +0.000, E1   -69.333, E3 +115906.510}
SPL {X  -135.354, Y  +761.800, Z    +0.000, E1   -68.789, E3 +115914.374}
SPL {X  -131.547, Y  +767.562, Z    +0.000, E1   -68.238, E3 +115921.543}
SPL {X  -127.113, Y  +773.655, Z    +0.000, E1   -67.565, E3 +115929.200}
SPL {X  -123.626, Y  +778.056, Z    +0.000, E1   -66.969, E3 +115934.760}
SPL {X   -86.110, Y  +811.340, Z    +0.000, E1   -55.142, E3 +116052.670}
ENDSPLINE

SPLINE
SPL {X  -126.688, Y  +774.208, Z    +0.000, E1   -50.278, E3 +116213.317}
SPL {X  -147.153, Y  +739.291, Z    +0.000, E1   -41.559, E3 +116234.152}
SPL {X  -156.578, Y  +709.366, Z    +0.000, E1   -27.394, E3 +116241.844}
SPL {X  -159.560, Y  +688.227, Z    +0.000, E1   -12.334, E3 +116244.409}
SPL {X  -159.987, Y  +677.470, Z    +0.000, E1    -2.943, E3 +116244.888}
SPL {X  -159.990, Y  +674.465, Z    +0.000, E1    +0.035, E3 +116244.921}
SPL {X  -159.990, Y  +672.210, Z    +0.000, E1    +4.112, E3 +116244.947}
SPL {X  -159.990, Y  +668.446, Z    +0.000, E1   +12.084, E3 +116245.073}
SPL {X  -159.990, Y  +663.424, Z    +0.000, E1   +23.273, E3 +116245.399}
SPL {X  -159.990, Y  +655.288, Z    +0.000, E1   +39.016, E3 +116246.288}
SPL {X  -159.990, Y  +641.020, Z    +0.000, E1   +55.512, E3 +116248.827}
SPL {X  -159.990, Y  +618.237, Z    +0.000, E1   +65.205, E3 +116255.352}
SPL {X  -159.990, Y  +545.807, Z    +0.000, E1   +71.095, E3 +116284.405}
SPL {X  -159.990, Y  +417.971, Z    +0.000, E1   +72.138, E3 +116353.065}
SPL {X  -147.674, Y  +315.943, Z    +0.000, E1   +77.803, E3 +116344.796}
ENDSPLINE

SPLINE
SPL {X  -149.193, Y  +319.722, Z    +0.000, E1   +76.912, E3 +116353.737}
ENDSPLINE

SPLINE
SPL {X  -149.153, Y  +319.620, Z    +0.000, E1   +75.840, E3 +116366.147}
ENDSPLINE

SPLINE
SPL {X  -149.679, Y  +320.993, Z    +0.000, E1   +74.493, E3 +116379.106}
SPL {X  -149.823, Y  +321.377, Z    +0.000, E1   +73.518, E3 +116388.464}
ENDSPLINE

SPLINE
SPL {X  -149.061, Y  +319.382, Z    +0.000, E1   +72.547, E3 +116398.706}
SPL {X  -148.522, Y  +318.020, Z    +0.000, E1   +71.446, E3 +116409.091}
SPL {X  -146.766, Y  +313.809, Z    +0.000, E1   +70.623, E3 +116418.743}
SPL {X  -143.180, Y  +306.112, Z    +0.000, E1   +70.169, E3 +116427.441}
SPL {X  -138.714, Y  +297.780, Z    +0.000, E1   +69.607, E3 +116437.187}
SPL {X  -135.202, Y  +291.959, Z    +0.000, E1   +69.085, E3 +116444.296}
SPL {X  -131.272, Y  +286.043, Z    +0.000, E1   +68.558, E3 +116451.535}
SPL {X  -127.436, Y  +280.769, Z    +0.000, E1   +67.934, E3 +116458.158}
SPL {X  -124.030, Y  +276.439, Z    +0.000, E1   +67.412, E3 +116463.522}
SPL {X   -89.505, Y  +244.889, Z    +0.000, E1   +58.168, E3 +116545.274}
ENDSPLINE

SPLINE
SPL {X  -111.763, Y  +263.019, Z    +0.000, E1   +52.505, E3 +116726.686}
SPL {X  -139.943, Y  +299.958, Z    +0.000, E1   +46.517, E3 +116761.026}
SPL {X  -152.249, Y  +328.336, Z    +0.000, E1   +36.404, E3 +116771.420}
SPL {X  -158.157, Y  +353.354, Z    +0.000, E1   +21.990, E3 +116776.144}
SPL {X  -159.630, Y  +366.769, Z    +0.000, E1   +11.595, E3 +116777.425}
SPL {X  -159.983, Y  +375.952, Z    +0.000, E1    +3.555, E3 +116777.806}
SPL {X  -159.990, Y  +379.545, Z    +0.000, E1    -0.045, E3 +116777.852}
SPL {X  -159.990, Y  +382.058, Z    +0.000, E1    -4.728, E3 +116777.884}
SPL {X  -159.990, Y  +387.492, Z    +0.000, E1   -16.478, E3 +116778.109}
SPL {X  -159.990, Y  +395.172, Z    +0.000, E1   -33.361, E3 +116778.736}
SPL {X  -159.990, Y  +405.626, Z    +0.000, E1   -49.217, E3 +116780.260}
SPL {X  -159.990, Y  +423.679, Z    +0.000, E1   -61.834, E3 +116784.531}
SPL {X  -159.990, Y  +491.183, Z    +0.000, E1   -70.406, E3 +116810.920}
SPL {X  -159.990, Y  +644.105, Z    +0.000, E1   -71.828, E3 +116895.489}
SPL {X  -159.990, Y  +665.410, Z    +0.000, E1   -71.813, E3 +116910.386}
SPL {X  -159.936, Y  +680.656, Z    +0.000, E1   -71.796, E3 +116921.104}
SPL {X  -158.712, Y  +696.685, Z    +0.000, E1   -71.696, E3 +116933.488}
SPL {X  -155.878, Y  +712.540, Z    +0.000, E1   -71.376, E3 +116947.505}
SPL {X  -152.746, Y  +724.097, Z    +0.000, E1   -71.019, E3 +116958.756}
SPL {X  -149.840, Y  +732.578, Z    +0.000, E1   -70.669, E3 +116967.582}
SPL {X  -147.044, Y  +739.548, Z    +0.000, E1   -70.332, E3 +116975.176}
SPL {X  -143.437, Y  +747.371, Z    +0.000, E1   -69.890, E3 +116984.040}
SPL {X  -139.209, Y  +755.353, Z    +0.000, E1   -69.333, E3 +116993.467}
SPL {X  -135.354, Y  +761.800, Z    +0.000, E1   -68.789, E3 +117001.330}
SPL {X  -131.547, Y  +767.562, Z    +0.000, E1   -68.238, E3 +117008.499}
SPL {X  -127.113, Y  +773.655, Z    +0.000, E1   -67.565, E3 +117016.156}
SPL {X  -123.626, Y  +778.056, Z    +0.000, E1   -66.969, E3 +117021.716}
SPL {X   -86.110, Y  +811.340, Z    +0.000, E1   -55.142, E3 +117139.627}
ENDSPLINE

SPLINE
SPL {X  -126.688, Y  +774.208, Z    +0.000, E1   -50.278, E3 +117300.274}
SPL {X  -147.153, Y  +739.291, Z    +0.000, E1   -41.559, E3 +117321.108}
SPL {X  -156.578, Y  +709.366, Z    +0.000, E1   -27.394, E3 +117328.801}
SPL {X  -159.560, Y  +688.227, Z    +0.000, E1   -12.334, E3 +117331.366}
SPL {X  -159.987, Y  +677.470, Z    +0.000, E1    -2.943, E3 +117331.845}
SPL {X  -159.990, Y  +674.465, Z    +0.000, E1    +0.035, E3 +117331.877}
SPL {X  -159.990, Y  +672.210, Z    +0.000, E1    +4.112, E3 +117331.904}
SPL {X  -159.990, Y  +668.446, Z    +0.000, E1   +12.084, E3 +117332.029}
SPL {X  -159.990, Y  +663.424, Z    +0.000, E1   +23.273, E3 +117332.356}
SPL {X  -159.990, Y  +655.288, Z    +0.000, E1   +39.016, E3 +117333.244}
SPL {X  -159.990, Y  +641.020, Z    +0.000, E1   +55.512, E3 +117335.784}
SPL {X  -159.990, Y  +618.237, Z    +0.000, E1   +65.205, E3 +117342.309}
SPL {X  -159.990, Y  +545.807, Z    +0.000, E1   +71.095, E3 +117371.362}
SPL {X  -159.990, Y  +417.971, Z    +0.000, E1   +72.138, E3 +117440.022}
SPL {X  -147.674, Y  +315.943, Z    +0.000, E1   +77.803, E3 +117431.752}
ENDSPLINE

SPLINE
SPL {X  -149.193, Y  +319.722, Z    +0.000, E1   +76.912, E3 +117440.694}
SPL {X  -149.265, Y  +319.910, Z    +0.000, E1   +76.148, E3 +117449.294}
ENDSPLINE

SPLINE
SPL {X  -149.092, Y  +319.462, Z    +0.000, E1   +75.437, E3 +117457.169}
ENDSPLINE

SPLINE
SPL {X  -149.679, Y  +320.993, Z    +0.000, E1   +74.493, E3 +117466.063}
SPL {X  -149.823, Y  +321.377, Z    +0.000, E1   +73.518, E3 +117475.421}
ENDSPLINE

SPLINE
SPL {X  -149.061, Y  +319.382, Z    +0.000, E1   +72.547, E3 +117485.662}
SPL {X  -148.522, Y  +318.020, Z    +0.000, E1   +71.446, E3 +117496.048}
SPL {X  -146.766, Y  +313.809, Z    +0.000, E1   +70.623, E3 +117505.700}
SPL {X  -143.180, Y  +306.112, Z    +0.000, E1   +70.169, E3 +117514.397}
SPL {X  -139.769, Y  +299.645, Z    +0.000, E1   +69.722, E3 +117521.964}
SPL {X  -136.083, Y  +293.369, Z    +0.000, E1   +69.227, E3 +117529.505}
SPL {X  -131.272, Y  +286.043, Z    +0.000, E1   +68.558, E3 +117538.491}
SPL {X  -126.312, Y  +279.306, Z    +0.000, E1   +67.784, E3 +117546.909}
SPL {X  -123.070, Y  +275.272, Z    +0.000, E1   +67.229, E3 +117551.947}
SPL {X   -89.505, Y  +244.889, Z    +0.000, E1   +58.168, E3 +117632.230}
ENDSPLINE

SPLINE
SPL {X  -111.763, Y  +263.019, Z    +0.000, E1   +52.505, E3 +117813.642}
SPL {X  -139.943, Y  +299.958, Z    +0.000, E1   +46.517, E3 +117847.983}
SPL {X  -152.249, Y  +328.336, Z    +0.000, E1   +36.404, E3 +117858.377}
SPL {X  -158.157, Y  +353.354, Z    +0.000, E1   +21.990, E3 +117863.100}
SPL {X  -159.828, Y  +370.311, Z    +0.000, E1    +8.652, E3 +117864.566}
SPL {X  -159.990, Y  +377.723, Z    +0.000, E1    +1.782, E3 +117864.797}
SPL {X  -159.990, Y  +379.545, Z    +0.000, E1    -0.045, E3 +117864.809}
SPL {X  -159.990, Y  +382.058, Z    +0.000, E1    -4.728, E3 +117864.841}
SPL {X  -159.990, Y  +387.492, Z    +0.000, E1   -16.478, E3 +117865.066}
SPL {X  -159.990, Y  +395.172, Z    +0.000, E1   -33.361, E3 +117865.693}
SPL {X  -159.990, Y  +403.640, Z    +0.000, E1   -46.960, E3 +117866.841}
SPL {X  -159.990, Y  +418.500, Z    +0.000, E1   -59.260, E3 +117870.196}
SPL {X  -159.990, Y  +491.183, Z    +0.000, E1   -70.406, E3 +117897.877}
SPL {X  -159.990, Y  +644.105, Z    +0.000, E1   -71.828, E3 +117982.445}
SPL {X  -159.990, Y  +665.410, Z    +0.000, E1   -71.813, E3 +117997.343}
SPL {X  -159.936, Y  +680.656, Z    +0.000, E1   -71.796, E3 +118008.061}
SPL {X  -158.712, Y  +696.685, Z    +0.000, E1   -71.696, E3 +118020.444}
SPL {X  -156.572, Y  +709.392, Z    +0.000, E1   -71.434, E3 +118031.591}
SPL {X  -154.409, Y  +718.389, Z    +0.000, E1   -71.209, E3 +118040.051}
SPL {X  -150.682, Y  +730.275, Z    +0.000, E1   -70.793, E3 +118052.050}
SPL {X  -147.044, Y  +739.548, Z    +0.000, E1   -70.332, E3 +118062.133}
SPL {X  -143.437, Y  +747.371, Z    +0.000, E1   -69.890, E3 +118070.996}
SPL {X  -139.209, Y  +755.353, Z    +0.000, E1   -69.333, E3 +118080.423}
SPL {X  -135.354, Y  +761.800, Z    +0.000, E1   -68.789, E3 +118088.287}
SPL {X  -131.547, Y  +767.562, Z    +0.000, E1   -68.238, E3 +118095.456}
SPL {X  -127.113, Y  +773.655, Z    +0.000, E1   -67.565, E3 +118103.113}
SPL {X  -123.626, Y  +778.056, Z    +0.000, E1   -66.969, E3 +118108.673}
SPL {X   -86.110, Y  +811.340, Z    +0.000, E1   -55.142, E3 +118226.583}
ENDSPLINE

SPLINE
SPL {X  -126.688, Y  +774.208, Z    +0.000, E1   -50.278, E3 +118387.230}
SPL {X  -147.153, Y  +739.291, Z    +0.000, E1   -41.559, E3 +118408.065}
SPL {X  -156.578, Y  +709.366, Z    +0.000, E1   -27.394, E3 +118415.758}
SPL {X  -159.560, Y  +688.227, Z    +0.000, E1   -12.334, E3 +118418.323}
SPL {X  -159.987, Y  +677.470, Z    +0.000, E1    -2.943, E3 +118418.801}
SPL {X  -159.990, Y  +674.465, Z    +0.000, E1    +0.035, E3 +118418.834}
SPL {X  -159.990, Y  +672.210, Z    +0.000, E1    +4.112, E3 +118418.860}
SPL {X  -159.990, Y  +668.446, Z    +0.000, E1   +12.084, E3 +118418.986}
SPL {X  -159.990, Y  +663.424, Z    +0.000, E1   +23.273, E3 +118419.312}
SPL {X  -159.990, Y  +655.288, Z    +0.000, E1   +39.016, E3 +118420.201}
SPL {X  -159.990, Y  +641.020, Z    +0.000, E1   +55.512, E3 +118422.740}
SPL {X  -159.990, Y  +618.237, Z    +0.000, E1   +65.205, E3 +118429.266}
SPL {X  -159.990, Y  +545.807, Z    +0.000, E1   +71.095, E3 +118458.318}
SPL {X  -159.990, Y  +417.971, Z    +0.000, E1   +72.138, E3 +118526.978}
SPL {X  -147.674, Y  +315.943, Z    +0.000, E1   +77.803, E3 +118518.709}
ENDSPLINE

SPLINE
SPL {X  -149.193, Y  +319.722, Z    +0.000, E1   +76.912, E3 +118527.650}
ENDSPLINE

SPLINE
SPL {X  -149.153, Y  +319.620, Z    +0.000, E1   +75.840, E3 +118540.060}
ENDSPLINE

SPLINE
SPL {X  -149.679, Y  +320.993, Z    +0.000, E1   +74.493, E3 +118553.019}
SPL {X  -149.823, Y  +321.377, Z    +0.000, E1   +73.518, E3 +118562.377}
ENDSPLINE

SPLINE
SPL {X  -149.061, Y  +319.382, Z    +0.000, E1   +72.547, E3 +118572.619}
SPL {X  -148.522, Y  +318.020, Z    +0.000, E1   +71.446, E3 +118583.004}
SPL {X  -146.766, Y  +313.809, Z    +0.000, E1   +70.623, E3 +118592.656}
SPL {X  -143.180, Y  +306.112, Z    +0.000, E1   +70.169, E3 +118601.354}
SPL {X  -139.769, Y  +299.645, Z    +0.000, E1   +69.722, E3 +118608.920}
SPL {X  -136.083, Y  +293.369, Z    +0.000, E1   +69.227, E3 +118616.462}
SPL {X  -132.274, Y  +287.498, Z    +0.000, E1   +68.678, E3 +118623.681}
SPL {X  -128.237, Y  +281.834, Z    +0.000, E1   +68.080, E3 +118630.717}
SPL {X  -125.186, Y  +277.874, Z    +0.000, E1   +67.573, E3 +118635.684}
SPL {X  -123.070, Y  +275.272, Z    +0.000, E1   +67.229, E3 +118638.904}
SPL {X   -89.505, Y  +244.889, Z    +0.000, E1   +58.168, E3 +118719.187}
ENDSPLINE

SPLINE
SPL {X  -111.763, Y  +263.019, Z    +0.000, E1   +52.505, E3 +118900.599}
SPL {X  -139.943, Y  +299.958, Z    +0.000, E1   +46.517, E3 +118934.939}
SPL {X  -154.122, Y  +334.569, Z    +0.000, E1   +33.405, E3 +118946.773}
SPL {X  -159.233, Y  +361.951, Z    +0.000, E1   +15.631, E3 +118950.952}
SPL {X  -159.983, Y  +375.952, Z    +0.000, E1    +3.555, E3 +118951.719}
SPL {X  -159.990, Y  +379.545, Z    +0.000, E1    -0.045, E3 +118951.765}
SPL {X  -159.990, Y  +382.058, Z    +0.000, E1    -4.728, E3 +118951.797}
SPL {X  -159.990, Y  +385.965, Z    +0.000, E1   -13.291, E3 +118951.932}
SPL {X  -159.990, Y  +391.054, Z    +0.000, E1   -24.765, E3 +118952.263}
SPL {X  -159.990, Y  +400.233, Z    +0.000, E1   -42.011, E3 +118953.308}
SPL {X  -159.990, Y  +418.500, Z    +0.000, E1   -59.260, E3 +118957.152}
SPL {X  -159.990, Y  +491.183, Z    +0.000, E1   -70.406, E3 +118984.834}
SPL {X  -159.990, Y  +644.105, Z    +0.000, E1   -71.828, E3 +119069.402}
SPL {X  -159.990, Y  +665.410, Z    +0.000, E1   -71.813, E3 +119084.299}
SPL {X  -159.784, Y  +684.619, Z    +0.000, E1   -71.795, E3 +119097.903}
SPL {X  -158.321, Y  +699.551, Z    +0.000, E1   -71.633, E3 +119109.855}
SPL {X  -155.878, Y  +712.540, Z    +0.000, E1   -71.376, E3 +119121.419}
SPL {X  -152.746, Y  +724.097, Z    +0.000, E1   -71.019, E3 +119132.669}
SPL {X  -149.840, Y  +732.578, Z    +0.000, E1   -70.669, E3 +119141.495}
SPL {X  -147.044, Y  +739.548, Z    +0.000, E1   -70.332, E3 +119149.089}
SPL {X  -143.437, Y  +747.371, Z    +0.000, E1   -69.890, E3 +119157.953}
SPL {X  -139.209, Y  +755.353, Z    +0.000, E1   -69.333, E3 +119167.380}
SPL {X  -135.354, Y  +761.800, Z    +0.000, E1   -68.789, E3 +119175.243}
SPL {X  -131.547, Y  +767.562, Z    +0.000, E1   -68.238, E3 +119182.412}
SPL {X  -127.113, Y  +773.655, Z    +0.000, E1   -67.565, E3 +119190.069}
SPL {X  -123.626, Y  +778.056, Z    +0.000, E1   -66.969, E3 +119195.629}
SPL {X   -86.110, Y  +811.340, Z    +0.000, E1   -55.142, E3 +119313.540}
ENDSPLINE

SPLINE
SPL {X  -126.688, Y  +774.208, Z    +0.000, E1   -50.278, E3 +119474.187}
SPL {X  -150.887, Y  +729.697, Z    +0.000, E1   -37.846, E3 +119498.043}
SPL {X  -157.603, Y  +704.031, Z    +0.000, E1   -23.939, E3 +119503.605}
SPL {X  -159.560, Y  +688.227, Z    +0.000, E1   -12.334, E3 +119505.279}
SPL {X  -159.987, Y  +677.470, Z    +0.000, E1    -2.943, E3 +119505.758}
SPL {X  -159.990, Y  +674.465, Z    +0.000, E1    +0.035, E3 +119505.790}
SPL {X  -159.990, Y  +672.210, Z    +0.000, E1    +4.112, E3 +119505.817}
SPL {X  -159.990, Y  +668.446, Z    +0.000, E1   +12.084, E3 +119505.942}
SPL {X  -159.990, Y  +663.424, Z    +0.000, E1   +23.273, E3 +119506.269}
SPL {X  -159.990, Y  +655.288, Z    +0.000, E1   +39.016, E3 +119507.157}
SPL {X  -159.990, Y  +641.020, Z    +0.000, E1   +55.512, E3 +119509.697}
SPL {X  -159.990, Y  +618.237, Z    +0.000, E1   +65.205, E3 +119516.222}
SPL {X  -159.990, Y  +545.807, Z    +0.000, E1   +71.095, E3 +119545.275}
SPL {X  -159.990, Y  +417.971, Z    +0.000, E1   +72.138, E3 +119613.935}
SPL {X  -147.674, Y  +315.943, Z    +0.000, E1   +77.803, E3 +119605.665}
ENDSPLINE

SPLINE
SPL {X  -149.193, Y  +319.722, Z    +0.000, E1   +76.912, E3 +119614.607}
SPL {X  -149.265, Y  +319.910, Z    +0.000, E1   +76.148, E3 +119623.207}
ENDSPLINE

SPLINE
SPL {X  -149.092, Y  +319.462, Z    +0.000, E1   +75.437, E3 +119631.082}
ENDSPLINE

SPLINE
SPL {X  -149.679, Y  +320.993, Z    +0.000, E1   +74.493, E3 +119639.976}
SPL {X  -149.823, Y  +321.377, Z    +0.000, E1   +73.518, E3 +119649.334}
ENDSPLINE

SPLINE
SPL {X  -149.061, Y  +319.382, Z    +0.000, E1   +72.547, E3 +119659.575}
SPL {X  -148.522, Y  +318.020, Z    +0.000, E1   +71.446, E3 +119669.961}
SPL {X  -146.766, Y  +313.809, Z    +0.000, E1   +70.623, E3 +119679.613}
SPL {X  -143.180, Y  +306.112, Z    +0.000, E1   +70.169, E3 +119688.310}
SPL {X  -139.769, Y  +299.645, Z    +0.000, E1   +69.722, E3 +119695.877}
SPL {X  -136.083, Y  +293.369, Z    +0.000, E1   +69.227, E3 +119703.418}
SPL {X  -131.272, Y  +286.043, Z    +0.000, E1   +68.558, E3 +119712.404}
SPL {X  -127.436, Y  +280.769, Z    +0.000, E1   +67.934, E3 +119719.028}
SPL {X  -124.030, Y  +276.439, Z    +0.000, E1   +67.412, E3 +119724.391}
SPL {X   -89.505, Y  +244.889, Z    +0.000, E1   +58.168, E3 +119806.143}
ENDSPLINE

SPLINE
SPL {X  -111.763, Y  +263.019, Z    +0.000, E1   +52.505, E3 +119987.555}
SPL {X  -139.943, Y  +299.958, Z    +0.000, E1   +46.517, E3 +120021.896}
SPL {X  -152.249, Y  +328.336, Z    +0.000, E1   +36.404, E3 +120032.290}
SPL {X  -158.157, Y  +353.354, Z    +0.000, E1   +21.990, E3 +120037.013}
SPL {X  -159.828, Y  +370.311, Z    +0.000, E1    +8.652, E3 +120038.479}
SPL {X  -159.990, Y  +379.415, Z    +0.000, E1    +0.198, E3 +120038.721}
SPL {X  -159.990, Y  +382.058, Z    +0.000, E1    -4.728, E3 +120038.754}
SPL {X  -159.990, Y  +387.492, Z    +0.000, E1   -16.478, E3 +120038.979}
SPL {X  -159.990, Y  +395.172, Z    +0.000, E1   -33.361, E3 +120039.606}
SPL {X  -159.990, Y  +403.640, Z    +0.000, E1   -46.960, E3 +120040.754}
SPL {X  -159.990, Y  +418.500, Z    +0.000, E1   -59.260, E3 +120044.109}
SPL {X  -159.990, Y  +491.183, Z    +0.000, E1   -70.406, E3 +120071.790}
SPL {X  -159.990, Y  +644.105, Z    +0.000, E1   -71.828, E3 +120156.358}
SPL {X  -159.990, Y  +665.410, Z    +0.000, E1   -71.813, E3 +120171.256}
SPL {X  -159.784, Y  +684.619, Z    +0.000, E1   -71.795, E3 +120184.860}
SPL {X  -158.321, Y  +699.551, Z    +0.000, E1   -71.633, E3 +120196.812}
SPL {X  -155.878, Y  +712.540, Z    +0.000, E1   -71.376, E3 +120208.375}
SPL {X  -152.746, Y  +724.097, Z    +0.000, E1   -71.019, E3 +120219.626}
SPL {X  -149.840, Y  +732.578, Z    +0.000, E1   -70.669, E3 +120228.452}
SPL {X  -147.044, Y  +739.548, Z    +0.000, E1   -70.332, E3 +120236.046}
SPL {X  -144.262, Y  +745.675, Z    +0.000, E1   -69.979, E3 +120242.984}
SPL {X  -141.227, Y  +751.679, Z    +0.000, E1   -69.593, E3 +120249.970}
SPL {X  -138.327, Y  +756.889, Z    +0.000, E1   -69.193, E3 +120256.221}
SPL {X  -134.311, Y  +763.433, Z    +0.000, E1   -68.667, E3 +120264.182}
SPL {X  -129.529, Y  +770.410, Z    +0.000, E1   -67.934, E3 +120272.946}
SPL {X  -126.163, Y  +774.886, Z    +0.000, E1   -67.384, E3 +120278.609}
SPL {X  -123.626, Y  +778.056, Z    +0.000, E1   -66.969, E3 +120282.586}
SPL {X   -86.110, Y  +811.340, Z    +0.000, E1   -55.142, E3 +120400.496}
ENDSPLINE

SPLINE
SPL {X  -126.688, Y  +774.208, Z    +0.000, E1   -50.278, E3 +120561.143}
SPL {X  -150.887, Y  +729.697, Z    +0.000, E1   -37.846, E3 +120584.999}
SPL {X  -157.603, Y  +704.031, Z    +0.000, E1   -23.939, E3 +120590.561}
SPL {X  -159.560, Y  +688.227, Z    +0.000, E1   -12.334, E3 +120592.236}
SPL {X  -159.987, Y  +677.470, Z    +0.000, E1    -2.943, E3 +120592.714}
SPL {X  -159.990, Y  +674.465, Z    +0.000, E1    +0.035, E3 +120592.747}
SPL {X  -159.990, Y  +672.210, Z    +0.000, E1    +4.112, E3 +120592.773}
SPL {X  -159.990, Y  +668.446, Z    +0.000, E1   +12.084, E3 +120592.899}
SPL {X  -159.990, Y  +663.424, Z    +0.000, E1   +23.273, E3 +120593.225}
SPL {X  -159.990, Y  +657.656, Z    +0.000, E1   +35.109, E3 +120593.786}
SPL {X  -159.990, Y  +651.328, Z    +0.000, E1   +45.171, E3 +120594.662}
SPL {X  -159.990, Y  +641.020, Z    +0.000, E1   +55.512, E3 +120596.653}
SPL {X  -159.990, Y  +618.237, Z    +0.000, E1   +65.205, E3 +120603.179}
SPL {X  -159.990, Y  +545.807, Z    +0.000, E1   +71.095, E3 +120632.231}
SPL {X  -159.990, Y  +417.971, Z    +0.000, E1   +72.138, E3 +120700.891}
SPL {X  -147.674, Y  +315.943, Z    +0.000, E1   +77.803, E3 +120692.622}
ENDSPLINE

SPLINE
SPL {X  -149.193, Y  +319.722, Z    +0.000, E1   +76.912, E3 +120701.564}
ENDSPLINE

SPLINE
SPL {X  -149.153, Y  +319.620, Z    +0.000, E1   +75.840, E3 +120713.973}
ENDSPLINE

SPLINE
SPL {X  -149.679, Y  +320.993, Z    +0.000, E1   +74.493, E3 +120726.933}
SPL {X  -149.823, Y  +321.377, Z    +0.000, E1   +73.518, E3 +120736.290}
ENDSPLINE

SPLINE
SPL {X  -149.061, Y  +319.382, Z    +0.000, E1   +72.547, E3 +120746.532}
SPL {X  -148.522, Y  +318.020, Z    +0.000, E1   +71.446, E3 +120756.917}
SPL {X  -146.766, Y  +313.809, Z    +0.000, E1   +70.623, E3 +120766.569}
SPL {X  -143.180, Y  +306.112, Z    +0.000, E1   +70.169, E3 +120775.267}
SPL {X  -139.769, Y  +299.645, Z    +0.000, E1   +69.722, E3 +120782.833}
SPL {X  -136.083, Y  +293.369, Z    +0.000, E1   +69.227, E3 +120790.375}
SPL {X  -132.274, Y  +287.498, Z    +0.000, E1   +68.678, E3 +120797.594}
SPL {X  -128.237, Y  +281.834, Z    +0.000, E1   +68.080, E3 +120804.630}
SPL {X  -125.186, Y  +277.874, Z    +0.000, E1   +67.573, E3 +120809.597}
SPL {X  -123.070, Y  +275.272, Z    +0.000, E1   +67.229, E3 +120812.817}
SPL {X   -89.505, Y  +244.889, Z    +0.000, E1   +58.168, E3 +120893.100}
ENDSPLINE

SPLINE
SPL {X  -111.763, Y  +263.019, Z    +0.000, E1   +52.505, E3 +121074.512}
SPL {X  -139.943, Y  +299.958, Z    +0.000, E1   +46.517, E3 +121108.852}
SPL {X  -154.122, Y  +334.569, Z    +0.000, E1   +33.405, E3 +121120.686}
SPL {X  -159.233, Y  +361.951, Z    +0.000, E1   +15.631, E3 +121124.865}
SPL {X  -159.983, Y  +375.952, Z    +0.000, E1    +3.555, E3 +121125.632}
SPL {X  -159.990, Y  +379.545, Z    +0.000, E1    -0.045, E3 +121125.678}
SPL {X  -159.990, Y  +382.058, Z    +0.000, E1    -4.728, E3 +121125.710}
SPL {X  -159.990, Y  +385.965, Z    +0.000, E1   -13.291, E3 +121125.845}
SPL {X  -159.990, Y  +391.054, Z    +0.000, E1   -24.765, E3 +121126.176}
SPL {X  -159.990, Y  +400.233, Z    +0.000, E1   -42.011, E3 +121127.221}
SPL {X  -159.990, Y  +418.500, Z    +0.000, E1   -59.260, E3 +121131.065}
SPL {X  -159.990, Y  +491.183, Z    +0.000, E1   -70.406, E3 +121158.747}
SPL {X  -159.990, Y  +644.105, Z    +0.000, E1   -71.828, E3 +121243.315}
SPL {X  -159.990, Y  +665.410, Z    +0.000, E1   -71.813, E3 +121258.213}
SPL {X  -159.784, Y  +684.619, Z    +0.000, E1   -71.795, E3 +121271.816}
SPL {X  -158.321, Y  +699.551, Z    +0.000, E1   -71.633, E3 +121283.768}
SPL {X  -155.878, Y  +712.540, Z    +0.000, E1   -71.376, E3 +121295.332}
SPL {X  -152.746, Y  +724.097, Z    +0.000, E1   -71.019, E3 +121306.583}
SPL {X  -149.840, Y  +732.578, Z    +0.000, E1   -70.669, E3 +121315.408}
SPL {X  -147.044, Y  +739.548, Z    +0.000, E1   -70.332, E3 +121323.002}
SPL {X  -143.437, Y  +747.371, Z    +0.000, E1   -69.890, E3 +121331.866}
SPL {X  -139.209, Y  +755.353, Z    +0.000, E1   -69.333, E3 +121341.293}
SPL {X  -135.354, Y  +761.800, Z    +0.000, E1   -68.789, E3 +121349.156}
SPL {X  -131.547, Y  +767.562, Z    +0.000, E1   -68.238, E3 +121356.326}
SPL {X  -128.543, Y  +771.755, Z    +0.000, E1   -67.757, E3 +121361.626}
SPL {X  -126.163, Y  +774.886, Z    +0.000, E1   -67.384, E3 +121365.566}
SPL {X  -123.626, Y  +778.056, Z    +0.000, E1   -66.969, E3 +121369.542}
SPL {X   -86.110, Y  +811.340, Z    +0.000, E1   -55.142, E3 +121487.453}
ENDSPLINE

SPLINE
SPL {X  -126.688, Y  +774.208, Z    +0.000, E1   -50.278, E3 +121648.100}
SPL {X  -150.887, Y  +729.697, Z    +0.000, E1   -37.846, E3 +121671.956}
SPL {X  -158.568, Y  +697.780, Z    +0.000, E1   -19.721, E3 +121678.286}
SPL {X  -159.967, Y  +679.234, Z    +0.000, E1    -4.684, E3 +121679.620}
SPL {X  -159.990, Y  +674.465, Z    +0.000, E1    +0.035, E3 +121679.703}
SPL {X  -159.990, Y  +672.210, Z    +0.000, E1    +4.112, E3 +121679.730}
SPL {X  -159.990, Y  +668.446, Z    +0.000, E1   +12.084, E3 +121679.855}
SPL {X  -159.990, Y  +663.424, Z    +0.000, E1   +23.273, E3 +121680.182}
SPL {X  -159.990, Y  +655.288, Z    +0.000, E1   +39.016, E3 +121681.070}
SPL {X  -159.990, Y  +641.020, Z    +0.000, E1   +55.512, E3 +121683.610}
SPL {X  -159.990, Y  +618.237, Z    +0.000, E1   +65.205, E3 +121690.135}
SPL {X  -159.990, Y  +545.807, Z    +0.000, E1   +71.095, E3 +121719.188}
SPL {X  -159.990, Y  +417.971, Z    +0.000, E1   +72.138, E3 +121787.848}
SPL {X  -147.674, Y  +315.943, Z    +0.000, E1   +77.803, E3 +121779.578}
ENDSPLINE

SPLINE
SPL {X  -149.193, Y  +319.722, Z    +0.000, E1   +76.912, E3 +121788.520}
ENDSPLINE

SPLINE
SPL {X  -149.153, Y  +319.620, Z    +0.000, E1   +75.840, E3 +121800.930}
ENDSPLINE

SPLINE
SPL {X  -149.679, Y  +320.993, Z    +0.000, E1   +74.493, E3 +121813.889}
SPL {X  -149.823, Y  +321.377, Z    +0.000, E1   +73.518, E3 +121823.247}
ENDSPLINE

SPLINE
SPL {X  -149.061, Y  +319.382, Z    +0.000, E1   +72.547, E3 +121833.488}
SPL {X  -148.201, Y  +317.223, Z    +0.000, E1   +71.184, E3 +121846.813}
SPL {X  -144.085, Y  +307.957, Z    +0.000, E1   +70.311, E3 +121860.059}
SPL {X  -139.769, Y  +299.645, Z    +0.000, E1   +69.722, E3 +121869.790}
SPL {X  -136.083, Y  +293.369, Z    +0.000, E1   +69.227, E3 +121877.331}
SPL {X  -131.272, Y  +286.043, Z    +0.000, E1   +68.558, E3 +121886.317}
SPL {X  -127.436, Y  +280.769, Z    +0.000, E1   +67.934, E3 +121892.941}
SPL {X  -124.030, Y  +276.439, Z    +0.000, E1   +67.412, E3 +121898.304}
SPL {X   -89.505, Y  +244.889, Z    +0.000, E1   +58.168, E3 +121980.057}
ENDSPLINE

SPLINE
SPL {X  -111.763, Y  +263.019, Z    +0.000, E1   +52.505, E3 +122161.468}
SPL {X  -139.943, Y  +299.958, Z    +0.000, E1   +46.517, E3 +122195.809}
SPL {X  -152.249, Y  +328.336, Z    +0.000, E1   +36.404, E3 +122206.203}
SPL {X  -158.157, Y  +353.354, Z    +0.000, E1   +21.990, E3 +122210.926}
SPL {X  -159.828, Y  +370.311, Z    +0.000, E1    +8.652, E3 +122212.392}
SPL {X  -159.990, Y  +377.723, Z    +0.000, E1    +1.782, E3 +122212.623}
SPL {X  -159.990, Y  +379.545, Z    +0.000, E1    -0.045, E3 +122212.635}
SPL {X  -159.990, Y  +382.058, Z    +0.000, E1    -4.728, E3 +122212.667}
SPL {X  -159.990, Y  +387.492, Z    +0.000, E1   -16.478, E3 +122212.892}
SPL {X  -159.990, Y  +395.172, Z    +0.000, E1   -33.361, E3 +122213.519}
SPL {X  -159.990, Y  +403.640, Z    +0.000, E1   -46.960, E3 +122214.667}
SPL {X  -159.990, Y  +418.500, Z    +0.000, E1   -59.260, E3 +122218.022}
SPL {X  -159.990, Y  +491.183, Z    +0.000, E1   -70.406, E3 +122245.703}
SPL {X  -159.990, Y  +636.738, Z    +0.000, E1   -71.802, E3 +122325.200}
SPL {X  -159.990, Y  +649.462, Z    +0.000, E1   -71.804, E3 +122334.070}
SPL {X  -159.990, Y  +665.410, Z    +0.000, E1   -71.813, E3 +122345.169}
SPL {X  -159.784, Y  +684.619, Z    +0.000, E1   -71.795, E3 +122358.773}
SPL {X  -158.321, Y  +699.551, Z    +0.000, E1   -71.633, E3 +122370.725}
SPL {X  -155.878, Y  +712.540, Z    +0.000, E1   -71.376, E3 +122382.288}
SPL {X  -152.746, Y  +724.097, Z    +0.000, E1   -71.019, E3 +122393.539}
SPL {X  -149.840, Y  +732.578, Z    +0.000, E1   -70.669, E3 +122402.365}
SPL {X  -147.044, Y  +739.548, Z    +0.000, E1   -70.332, E3 +122409.959}
SPL {X  -144.262, Y  +745.675, Z    +0.000, E1   -69.979, E3 +122416.897}
SPL {X  -141.227, Y  +751.679, Z    +0.000, E1   -69.593, E3 +122423.883}
SPL {X  -138.327, Y  +756.889, Z    +0.000, E1   -69.193, E3 +122430.134}
SPL {X  -135.354, Y  +761.800, Z    +0.000, E1   -68.789, E3 +122436.113}
SPL {X  -131.547, Y  +767.562, Z    +0.000, E1   -68.238, E3 +122443.282}
SPL {X  -128.543, Y  +771.755, Z    +0.000, E1   -67.757, E3 +122448.583}
SPL {X  -126.163, Y  +774.886, Z    +0.000, E1   -67.384, E3 +122452.522}
SPL {X  -123.626, Y  +778.056, Z    +0.000, E1   -66.969, E3 +122456.499}
SPL {X   -86.110, Y  +811.340, Z    +0.000, E1   -55.142, E3 +122574.409}
ENDSPLINE

SPLINE
SPL {X  -126.688, Y  +774.208, Z    +0.000, E1   -50.278, E3 +122735.056}
SPL {X  -150.887, Y  +729.697, Z    +0.000, E1   -37.846, E3 +122758.912}
SPL {X  -158.568, Y  +697.780, Z    +0.000, E1   -19.721, E3 +122765.242}
SPL {X  -159.967, Y  +679.234, Z    +0.000, E1    -4.684, E3 +122766.577}
SPL {X  -159.990, Y  +674.465, Z    +0.000, E1    +0.035, E3 +122766.660}
SPL {X  -159.990, Y  +672.210, Z    +0.000, E1    +4.112, E3 +122766.686}
SPL {X  -159.990, Y  +668.446, Z    +0.000, E1   +12.084, E3 +122766.812}
SPL {X  -159.990, Y  +663.424, Z    +0.000, E1   +23.273, E3 +122767.138}
SPL {X  -159.990, Y  +655.288, Z    +0.000, E1   +39.016, E3 +122768.027}
SPL {X  -159.990, Y  +641.020, Z    +0.000, E1   +55.512, E3 +122770.566}
SPL {X  -159.990, Y  +618.237, Z    +0.000, E1   +65.205, E3 +122777.092}
SPL {X  -159.990, Y  +545.807, Z    +0.000, E1   +71.095, E3 +122806.144}
SPL {X  -159.990, Y  +417.971, Z    +0.000, E1   +72.138, E3 +122874.804}
SPL {X  -147.674, Y  +315.943, Z    +0.000, E1   +77.803, E3 +122866.535}
ENDSPLINE

SPLINE
SPL {X  -149.193, Y  +319.722, Z    +0.000, E1   +76.912, E3 +122875.477}
ENDSPLINE

SPLINE
SPL {X  -149.153, Y  +319.620, Z    +0.000, E1   +75.840, E3 +122887.886}
ENDSPLINE

SPLINE
SPL {X  -149.679, Y  +320.993, Z    +0.000, E1   +74.493, E3 +122900.846}
SPL {X  -149.823, Y  +321.377, Z    +0.000, E1   +73.518, E3 +122910.203}
ENDSPLINE

SPLINE
SPL {X  -149.061, Y  +319.382, Z    +0.000, E1   +72.547, E3 +122920.445}
SPL {X  -148.201, Y  +317.223, Z    +0.000, E1   +71.184, E3 +122933.769}
SPL {X  -144.085, Y  +307.957, Z    +0.000, E1   +70.311, E3 +122947.016}
SPL {X  -139.769, Y  +299.645, Z    +0.000, E1   +69.722, E3 +122956.747}
SPL {X  -136.083, Y  +293.369, Z    +0.000, E1   +69.227, E3 +122964.288}
SPL {X  -131.272, Y  +286.043, Z    +0.000, E1   +68.558, E3 +122973.274}
SPL {X  -127.436, Y  +280.769, Z    +0.000, E1   +67.934, E3 +122979.897}
SPL {X  -124.030, Y  +276.439, Z    +0.000, E1   +67.412, E3 +122985.261}
SPL {X   -89.505, Y  +244.889, Z    +0.000, E1   +58.168, E3 +123067.013}
ENDSPLINE

SPLINE
SPL {X  -111.763, Y  +263.019, Z    +0.000, E1   +52.505, E3 +123248.425}
SPL {X  -139.943, Y  +299.958, Z    +0.000, E1   +46.517, E3 +123282.765}
SPL {X  -154.122, Y  +334.569, Z    +0.000, E1   +33.405, E3 +123294.600}
SPL {X  -159.233, Y  +361.951, Z    +0.000, E1   +15.631, E3 +123298.778}
SPL {X  -159.983, Y  +375.952, Z    +0.000, E1    +3.555, E3 +123299.545}
SPL {X  -159.990, Y  +379.545, Z    +0.000, E1    -0.045, E3 +123299.591}
SPL {X  -159.990, Y  +382.058, Z    +0.000, E1    -4.728, E3 +123299.623}
SPL {X  -159.990, Y  +387.492, Z    +0.000, E1   -16.478, E3 +123299.848}
SPL {X  -159.990, Y  +395.172, Z    +0.000, E1   -33.361, E3 +123300.475}
SPL {X  -159.990, Y  +405.626, Z    +0.000, E1   -49.217, E3 +123301.999}
SPL {X  -159.990, Y  +423.679, Z    +0.000, E1   -61.834, E3 +123306.270}
SPL {X  -159.990, Y  +491.183, Z    +0.000, E1   -70.406, E3 +123332.660}
SPL {X  -159.990, Y  +644.105, Z    +0.000, E1   -71.828, E3 +123417.228}
SPL {X  -159.990, Y  +665.410, Z    +0.000, E1   -71.813, E3 +123432.126}
SPL {X  -159.784, Y  +684.619, Z    +0.000, E1   -71.795, E3 +123445.729}
SPL {X  -158.321, Y  +699.551, Z    +0.000, E1   -71.633, E3 +123457.681}
SPL {X  -155.878, Y  +712.540, Z    +0.000, E1   -71.376, E3 +123469.245}
SPL {X  -152.746, Y  +724.097, Z    +0.000, E1   -71.019, E3 +123480.496}
SPL {X  -149.840, Y  +732.578, Z    +0.000, E1   -70.669, E3 +123489.321}
SPL {X  -147.044, Y  +739.548, Z    +0.000, E1   -70.332, E3 +123496.915}
SPL {X  -143.437, Y  +747.371, Z    +0.000, E1   -69.890, E3 +123505.779}
SPL {X  -139.209, Y  +755.353, Z    +0.000, E1   -69.333, E3 +123515.206}
SPL {X  -134.311, Y  +763.433, Z    +0.000, E1   -68.667, E3 +123525.052}
SPL {X  -129.529, Y  +770.410, Z    +0.000, E1   -67.934, E3 +123533.816}
SPL {X  -126.163, Y  +774.886, Z    +0.000, E1   -67.384, E3 +123539.479}
SPL {X  -123.626, Y  +778.056, Z    +0.000, E1   -66.969, E3 +123543.455}
SPL {X   -86.110, Y  +811.340, Z    +0.000, E1   -55.142, E3 +123661.366}
ENDSPLINE

SPLINE
SPL {X  -126.688, Y  +774.208, Z    +0.000, E1   -50.278, E3 +123822.013}
SPL {X  -150.887, Y  +729.697, Z    +0.000, E1   -37.846, E3 +123845.869}
SPL {X  -158.568, Y  +697.780, Z    +0.000, E1   -19.721, E3 +123852.199}
SPL {X  -159.967, Y  +679.234, Z    +0.000, E1    -4.684, E3 +123853.533}
SPL {X  -159.990, Y  +674.465, Z    +0.000, E1    +0.035, E3 +123853.616}
SPL {X  -159.990, Y  +672.210, Z    +0.000, E1    +4.112, E3 +123853.643}
SPL {X  -159.990, Y  +668.446, Z    +0.000, E1   +12.084, E3 +123853.768}
SPL {X  -159.990, Y  +663.424, Z    +0.000, E1   +23.273, E3 +123854.095}
SPL {X  -159.990, Y  +655.288, Z    +0.000, E1   +39.016, E3 +123854.983}
SPL {X  -159.990, Y  +641.020, Z    +0.000, E1   +55.512, E3 +123857.523}
SPL {X  -159.990, Y  +618.237, Z    +0.000, E1   +65.205, E3 +123864.048}
SPL {X  -159.990, Y  +545.807, Z    +0.000, E1   +71.095, E3 +123893.101}
SPL {X  -159.990, Y  +417.971, Z    +0.000, E1   +72.138, E3 +123961.761}
SPL {X  -147.674, Y  +315.943, Z    +0.000, E1   +77.803, E3 +123953.491}
ENDSPLINE

SPLINE
SPL {X  -149.193, Y  +319.722, Z    +0.000, E1   +76.912, E3 +123962.433}
ENDSPLINE

SPLINE
SPL {X  -149.153, Y  +319.620, Z    +0.000, E1   +75.840, E3 +123974.843}
ENDSPLINE

SPLINE
SPL {X  -149.679, Y  +320.993, Z    +0.000, E1   +74.493, E3 +123987.802}
SPL {X  -149.823, Y  +321.377, Z    +0.000, E1   +73.518, E3 +123997.160}
ENDSPLINE

SPLINE
SPL {X  -149.061, Y  +319.382, Z    +0.000, E1   +72.547, E3 +124007.401}
SPL {X  -148.201, Y  +317.223, Z    +0.000, E1   +71.184, E3 +124020.726}
SPL {X  -144.085, Y  +307.957, Z    +0.000, E1   +70.311, E3 +124033.972}
SPL {X  -139.769, Y  +299.645, Z    +0.000, E1   +69.722, E3 +124043.703}
SPL {X  -136.083, Y  +293.369, Z    +0.000, E1   +69.227, E3 +124051.244}
SPL {X  -131.272, Y  +286.043, Z    +0.000, E1   +68.558, E3 +124060.231}
SPL {X  -127.436, Y  +280.769, Z    +0.000, E1   +67.934, E3 +124066.854}
SPL {X  -124.030, Y  +276.439, Z    +0.000, E1   +67.412, E3 +124072.217}
SPL {X   -89.505, Y  +244.889, Z    +0.000, E1   +58.168, E3 +124153.970}
ENDSPLINE

SPLINE
SPL {X  -111.763, Y  +263.019, Z    +0.000, E1   +52.505, E3 +124335.381}
SPL {X  -139.943, Y  +299.958, Z    +0.000, E1   +46.517, E3 +124369.722}
SPL {X  -152.249, Y  +328.336, Z    +0.000, E1   +36.404, E3 +124380.116}
SPL {X  -158.157, Y  +353.354, Z    +0.000, E1   +21.990, E3 +124384.839}
SPL {X  -159.828, Y  +370.311, Z    +0.000, E1    +8.652, E3 +124386.305}
SPL {X  -159.990, Y  +377.723, Z    +0.000, E1    +1.782, E3 +124386.536}
SPL {X  -159.990, Y  +379.545, Z    +0.000, E1    -0.045, E3 +124386.548}
SPL {X  -159.990, Y  +382.058, Z    +0.000, E1    -4.728, E3 +124386.580}
SPL {X  -159.990, Y  +387.492, Z    +0.000, E1   -16.478, E3 +124386.805}
SPL {X  -159.990, Y  +395.172, Z    +0.000, E1   -33.361, E3 +124387.432}
SPL {X  -159.990, Y  +403.640, Z    +0.000, E1   -46.960, E3 +124388.580}
SPL {X  -159.990, Y  +418.500, Z    +0.000, E1   -59.260, E3 +124391.935}
SPL {X  -159.990, Y  +491.183, Z    +0.000, E1   -70.406, E3 +124419.616}
SPL {X  -159.990, Y  +636.738, Z    +0.000, E1   -71.802, E3 +124499.114}
SPL {X  -159.990, Y  +649.462, Z    +0.000, E1   -71.804, E3 +124507.983}
SPL {X  -159.990, Y  +665.410, Z    +0.000, E1   -71.813, E3 +124519.082}
SPL {X  -159.784, Y  +684.619, Z    +0.000, E1   -71.795, E3 +124532.686}
SPL {X  -158.321, Y  +699.551, Z    +0.000, E1   -71.633, E3 +124544.638}
SPL {X  -155.878, Y  +712.540, Z    +0.000, E1   -71.376, E3 +124556.201}
SPL {X  -152.746, Y  +724.097, Z    +0.000, E1   -71.019, E3 +124567.452}
SPL {X  -149.840, Y  +732.578, Z    +0.000, E1   -70.669, E3 +124576.278}
SPL {X  -147.044, Y  +739.548, Z    +0.000, E1   -70.332, E3 +124583.872}
SPL {X  -144.262, Y  +745.675, Z    +0.000, E1   -69.979, E3 +124590.810}
SPL {X  -141.227, Y  +751.679, Z    +0.000, E1   -69.593, E3 +124597.796}
SPL {X  -138.327, Y  +756.889, Z    +0.000, E1   -69.193, E3 +124604.047}
SPL {X  -135.354, Y  +761.800, Z    +0.000, E1   -68.789, E3 +124610.026}
SPL {X  -131.547, Y  +767.562, Z    +0.000, E1   -68.238, E3 +124617.195}
SPL {X  -128.543, Y  +771.755, Z    +0.000, E1   -67.757, E3 +124622.496}
SPL {X  -126.163, Y  +774.886, Z    +0.000, E1   -67.384, E3 +124626.435}
SPL {X  -123.626, Y  +778.056, Z    +0.000, E1   -66.969, E3 +124630.412}
SPL {X   -86.110, Y  +811.340, Z    +0.000, E1   -55.142, E3 +124748.322}
ENDSPLINE

SPLINE
SPL {X  -126.688, Y  +774.208, Z    +0.000, E1   -50.278, E3 +124908.969}
SPL {X  -150.887, Y  +729.697, Z    +0.000, E1   -37.846, E3 +124932.825}
SPL {X  -158.568, Y  +697.780, Z    +0.000, E1   -19.721, E3 +124939.155}
SPL {X  -159.967, Y  +679.234, Z    +0.000, E1    -4.684, E3 +124940.490}
SPL {X  -159.990, Y  +674.465, Z    +0.000, E1    +0.035, E3 +124940.573}
SPL {X  -159.990, Y  +672.210, Z    +0.000, E1    +4.112, E3 +124940.599}
SPL {X  -159.990, Y  +668.446, Z    +0.000, E1   +12.084, E3 +124940.725}
SPL {X  -159.990, Y  +663.424, Z    +0.000, E1   +23.273, E3 +124941.051}
SPL {X  -159.990, Y  +655.288, Z    +0.000, E1   +39.016, E3 +124941.940}
SPL {X  -159.990, Y  +641.020, Z    +0.000, E1   +55.512, E3 +124944.479}
SPL {X  -159.990, Y  +618.237, Z    +0.000, E1   +65.205, E3 +124951.005}
SPL {X  -159.990, Y  +545.807, Z    +0.000, E1   +71.095, E3 +124980.057}
SPL {X  -159.990, Y  +417.971, Z    +0.000, E1   +72.138, E3 +125048.717}
SPL {X  -147.674, Y  +315.943, Z    +0.000, E1   +77.803, E3 +125040.448}
ENDSPLINE

SPLINE
SPL {X  -149.193, Y  +319.722, Z    +0.000, E1   +76.912, E3 +125049.390}
SPL {X  -149.265, Y  +319.910, Z    +0.000, E1   +76.148, E3 +125057.990}
ENDSPLINE

SPLINE
SPL {X  -149.092, Y  +319.462, Z    +0.000, E1   +75.437, E3 +125065.865}
ENDSPLINE

SPLINE
SPL {X  -149.679, Y  +320.993, Z    +0.000, E1   +74.493, E3 +125074.759}
SPL {X  -149.823, Y  +321.377, Z    +0.000, E1   +73.518, E3 +125084.116}
ENDSPLINE

SPLINE
SPL {X  -149.061, Y  +319.382, Z    +0.000, E1   +72.547, E3 +125094.358}
SPL {X  -148.522, Y  +318.020, Z    +0.000, E1   +71.446, E3 +125104.743}
SPL {X  -146.766, Y  +313.809, Z    +0.000, E1   +70.623, E3 +125114.395}
SPL {X  -143.180, Y  +306.112, Z    +0.000, E1   +70.169, E3 +125123.093}
SPL {X  -138.714, Y  +297.780, Z    +0.000, E1   +69.607, E3 +125132.839}
SPL {X  -135.202, Y  +291.959, Z    +0.000, E1   +69.085, E3 +125139.948}
SPL {X  -131.272, Y  +286.043, Z    +0.000, E1   +68.558, E3 +125147.187}
SPL {X  -127.436, Y  +280.769, Z    +0.000, E1   +67.934, E3 +125153.810}
SPL {X  -124.030, Y  +276.439, Z    +0.000, E1   +67.412, E3 +125159.174}
SPL {X   -89.505, Y  +244.889, Z    +0.000, E1   +58.168, E3 +125240.926}
ENDSPLINE

SPLINE
SPL {X  -111.763, Y  +263.019, Z    +0.000, E1   +52.505, E3 +125422.338}
SPL {X  -139.943, Y  +299.958, Z    +0.000, E1   +46.517, E3 +125456.678}
SPL {X  -152.249, Y  +328.336, Z    +0.000, E1   +36.404, E3 +125467.072}
SPL {X  -158.157, Y  +353.354, Z    +0.000, E1   +21.990, E3 +125471.796}
SPL {X  -159.828, Y  +370.311, Z    +0.000, E1    +8.652, E3 +125473.261}
SPL {X  -159.990, Y  +377.723, Z    +0.000, E1    +1.782, E3 +125473.492}
SPL {X  -159.990, Y  +379.545, Z    +0.000, E1    -0.045, E3 +125473.504}
SPL {X  -159.990, Y  +382.058, Z    +0.000, E1    -4.728, E3 +125473.536}
SPL {X  -159.990, Y  +385.965, Z    +0.000, E1   -13.291, E3 +125473.671}
SPL {X  -159.990, Y  +391.054, Z    +0.000, E1   -24.765, E3 +125474.002}
SPL {X  -159.990, Y  +400.233, Z    +0.000, E1   -42.011, E3 +125475.047}
SPL {X  -159.990, Y  +418.500, Z    +0.000, E1   -59.260, E3 +125478.891}
SPL {X  -159.990, Y  +491.183, Z    +0.000, E1   -70.406, E3 +125506.573}
SPL {X  -159.990, Y  +644.105, Z    +0.000, E1   -71.828, E3 +125591.141}
SPL {X  -159.990, Y  +665.410, Z    +0.000, E1   -71.813, E3 +125606.039}
SPL {X  -159.936, Y  +680.656, Z    +0.000, E1   -71.796, E3 +125616.756}
SPL {X  -158.712, Y  +696.685, Z    +0.000, E1   -71.696, E3 +125629.140}
SPL {X  -155.878, Y  +712.540, Z    +0.000, E1   -71.376, E3 +125643.158}
SPL {X  -152.746, Y  +724.097, Z    +0.000, E1   -71.019, E3 +125654.409}
SPL {X  -149.840, Y  +732.578, Z    +0.000, E1   -70.669, E3 +125663.234}
SPL {X  -147.044, Y  +739.548, Z    +0.000, E1   -70.332, E3 +125670.828}
SPL {X  -143.437, Y  +747.371, Z    +0.000, E1   -69.890, E3 +125679.692}
SPL {X  -139.209, Y  +755.353, Z    +0.000, E1   -69.333, E3 +125689.119}
SPL {X  -135.354, Y  +761.800, Z    +0.000, E1   -68.789, E3 +125696.983}
SPL {X  -131.547, Y  +767.562, Z    +0.000, E1   -68.238, E3 +125704.152}
SPL {X  -127.113, Y  +773.655, Z    +0.000, E1   -67.565, E3 +125711.808}
SPL {X  -123.626, Y  +778.056, Z    +0.000, E1   -66.969, E3 +125717.368}
SPL {X   -86.110, Y  +811.340, Z    +0.000, E1   -55.142, E3 +125835.279}
ENDSPLINE

SPLINE
SPL {X  -126.688, Y  +774.208, Z    +0.000, E1   -50.278, E3 +125995.926}
SPL {X  -147.153, Y  +739.291, Z    +0.000, E1   -41.559, E3 +126016.761}
SPL {X  -156.578, Y  +709.366, Z    +0.000, E1   -27.394, E3 +126024.453}
SPL {X  -159.560, Y  +688.227, Z    +0.000, E1   -12.334, E3 +126027.018}
SPL {X  -159.987, Y  +677.470, Z    +0.000, E1    -2.943, E3 +126027.497}
SPL {X  -159.990, Y  +674.465, Z    +0.000, E1    +0.035, E3 +126027.529}
SPL {X  -159.990, Y  +672.210, Z    +0.000, E1    +4.112, E3 +126027.556}
SPL {X  -159.990, Y  +668.446, Z    +0.000, E1   +12.084, E3 +126027.681}
SPL {X  -159.990, Y  +663.424, Z    +0.000, E1   +23.273, E3 +126028.008}
SPL {X  -159.990, Y  +655.288, Z    +0.000, E1   +39.016, E3 +126028.897}
SPL {X  -159.990, Y  +641.020, Z    +0.000, E1   +55.512, E3 +126031.436}
SPL {X  -159.990, Y  +618.237, Z    +0.000, E1   +65.205, E3 +126037.961}
SPL {X  -159.990, Y  +545.807, Z    +0.000, E1   +71.095, E3 +126067.014}
SPL {X  -149.334, Y  +320.087, Z    +0.000, E1   +77.218, E3 +126132.833}
SPL {X  -149.265, Y  +319.910, Z    +0.000, E1   +76.148, E3 +126144.946}
SPL {X  -149.092, Y  +319.462, Z    +0.000, E1   +75.437, E3 +126152.821}
ENDSPLINE

SPLINE
SPL {X  -149.679, Y  +320.993, Z    +0.000, E1   +74.493, E3 +126161.715}
SPL {X  -149.823, Y  +321.377, Z    +0.000, E1   +73.518, E3 +126171.073}
ENDSPLINE

SPLINE
SPL {X  -149.061, Y  +319.382, Z    +0.000, E1   +72.547, E3 +126181.314}
SPL {X  -148.522, Y  +318.020, Z    +0.000, E1   +71.446, E3 +126191.700}
SPL {X  -146.766, Y  +313.809, Z    +0.000, E1   +70.623, E3 +126201.352}
SPL {X  -143.180, Y  +306.112, Z    +0.000, E1   +70.169, E3 +126210.049}
SPL {X  -139.769, Y  +299.645, Z    +0.000, E1   +69.722, E3 +126217.616}
SPL {X  -136.083, Y  +293.369, Z    +0.000, E1   +69.227, E3 +126225.157}
SPL {X  -132.274, Y  +287.498, Z    +0.000, E1   +68.678, E3 +126232.377}
SPL {X  -128.237, Y  +281.834, Z    +0.000, E1   +68.080, E3 +126239.413}
SPL {X  -124.030, Y  +276.439, Z    +0.000, E1   +67.412, E3 +126246.130}
SPL {X   -89.505, Y  +244.889, Z    +0.000, E1   +58.168, E3 +126327.883}
ENDSPLINE

SPLINE
SPL {X  -111.763, Y  +263.019, Z    +0.000, E1   +52.505, E3 +126509.295}
SPL {X  -139.943, Y  +299.958, Z    +0.000, E1   +46.517, E3 +126543.635}
SPL {X  -154.122, Y  +334.569, Z    +0.000, E1   +33.405, E3 +126555.469}
SPL {X  -159.233, Y  +361.951, Z    +0.000, E1   +15.631, E3 +126559.648}
SPL {X  -159.983, Y  +375.952, Z    +0.000, E1    +3.555, E3 +126560.414}
SPL {X  -159.990, Y  +379.545, Z    +0.000, E1    -0.045, E3 +126560.461}
SPL {X  -159.990, Y  +382.058, Z    +0.000, E1    -4.728, E3 +126560.493}
SPL {X  -159.990, Y  +387.492, Z    +0.000, E1   -16.478, E3 +126560.718}
SPL {X  -159.990, Y  +395.172, Z    +0.000, E1   -33.361, E3 +126561.345}
SPL {X  -159.990, Y  +405.626, Z    +0.000, E1   -49.217, E3 +126562.868}
SPL {X  -159.990, Y  +423.679, Z    +0.000, E1   -61.834, E3 +126567.140}
SPL {X  -159.990, Y  +491.183, Z    +0.000, E1   -70.406, E3 +126593.529}
SPL {X  -159.990, Y  +644.105, Z    +0.000, E1   -71.828, E3 +126678.097}
SPL {X  -159.990, Y  +665.410, Z    +0.000, E1   -71.813, E3 +126692.995}
SPL {X  -159.936, Y  +680.656, Z    +0.000, E1   -71.796, E3 +126703.713}
SPL {X  -158.712, Y  +696.685, Z    +0.000, E1   -71.696, E3 +126716.096}
SPL {X  -156.572, Y  +709.392, Z    +0.000, E1   -71.434, E3 +126727.244}
SPL {X  -154.409, Y  +718.389, Z    +0.000, E1   -71.209, E3 +126735.703}
SPL {X  -150.682, Y  +730.275, Z    +0.000, E1   -70.793, E3 +126747.702}
SPL {X  -147.044, Y  +739.548, Z    +0.000, E1   -70.332, E3 +126757.785}
SPL {X  -144.262, Y  +745.675, Z    +0.000, E1   -69.979, E3 +126764.723}
SPL {X  -141.227, Y  +751.679, Z    +0.000, E1   -69.593, E3 +126771.709}
SPL {X  -138.327, Y  +756.889, Z    +0.000, E1   -69.193, E3 +126777.960}
SPL {X  -135.354, Y  +761.800, Z    +0.000, E1   -68.789, E3 +126783.939}
SPL {X  -131.547, Y  +767.562, Z    +0.000, E1   -68.238, E3 +126791.108}
SPL {X  -127.113, Y  +773.655, Z    +0.000, E1   -67.565, E3 +126798.765}
SPL {X  -123.626, Y  +778.056, Z    +0.000, E1   -66.969, E3 +126804.325}
SPL {X   -86.110, Y  +811.340, Z    +0.000, E1   -55.142, E3 +126922.235}
ENDSPLINE

SPLINE
SPL {X  -126.688, Y  +774.208, Z    +0.000, E1   -50.278, E3 +127082.882}
SPL {X  -147.153, Y  +739.291, Z    +0.000, E1   -41.559, E3 +127103.717}
SPL {X  -156.578, Y  +709.366, Z    +0.000, E1   -27.394, E3 +127111.410}
SPL {X  -159.560, Y  +688.227, Z    +0.000, E1   -12.334, E3 +127113.975}
SPL {X  -159.987, Y  +677.470, Z    +0.000, E1    -2.943, E3 +127114.453}
SPL {X  -159.990, Y  +674.465, Z    +0.000, E1    +0.035, E3 +127114.486}
SPL {X  -159.990, Y  +672.210, Z    +0.000, E1    +4.112, E3 +127114.512}
SPL {X  -159.990, Y  +668.446, Z    +0.000, E1   +12.084, E3 +127114.638}
SPL {X  -159.990, Y  +663.424, Z    +0.000, E1   +23.273, E3 +127114.964}
SPL {X  -159.990, Y  +655.288, Z    +0.000, E1   +39.016, E3 +127115.853}
SPL {X  -159.990, Y  +641.020, Z    +0.000, E1   +55.512, E3 +127118.392}
SPL {X  -159.990, Y  +618.237, Z    +0.000, E1   +65.205, E3 +127124.918}
SPL {X  -159.990, Y  +545.807, Z    +0.000, E1   +71.095, E3 +127153.971}
SPL {X  -159.990, Y  +417.971, Z    +0.000, E1   +72.138, E3 +127222.630}
SPL {X  -147.674, Y  +315.943, Z    +0.000, E1   +77.803, E3 +127214.361}
ENDSPLINE

SPLINE
SPL {X  -149.193, Y  +319.722, Z    +0.000, E1   +76.912, E3 +127223.303}
ENDSPLINE

SPLINE
SPL {X  -149.153, Y  +319.620, Z    +0.000, E1   +75.840, E3 +127235.712}
ENDSPLINE

SPLINE
SPL {X  -149.679, Y  +320.993, Z    +0.000, E1   +74.493, E3 +127248.672}
SPL {X  -149.823, Y  +321.377, Z    +0.000, E1   +73.518, E3 +127258.029}
ENDSPLINE

SPLINE
SPL {X  -149.061, Y  +319.382, Z    +0.000, E1   +72.547, E3 +127268.271}
SPL {X  -148.522, Y  +318.020, Z    +0.000, E1   +71.446, E3 +127278.656}
SPL {X  -146.766, Y  +313.809, Z    +0.000, E1   +70.623, E3 +127288.308}
SPL {X  -143.180, Y  +306.112, Z    +0.000, E1   +70.169, E3 +127297.006}
SPL {X  -139.769, Y  +299.645, Z    +0.000, E1   +69.722, E3 +127304.573}
SPL {X  -136.083, Y  +293.369, Z    +0.000, E1   +69.227, E3 +127312.114}
SPL {X  -132.274, Y  +287.498, Z    +0.000, E1   +68.678, E3 +127319.333}
SPL {X  -128.237, Y  +281.834, Z    +0.000, E1   +68.080, E3 +127326.370}
SPL {X  -124.030, Y  +276.439, Z    +0.000, E1   +67.412, E3 +127333.087}
SPL {X   -89.505, Y  +244.889, Z    +0.000, E1   +58.168, E3 +127414.839}
ENDSPLINE

SPLINE
SPL {X  -111.763, Y  +263.019, Z    +0.000, E1   +52.505, E3 +127596.251}
SPL {X  -139.943, Y  +299.958, Z    +0.000, E1   +46.517, E3 +127630.591}
SPL {X  -154.122, Y  +334.569, Z    +0.000, E1   +33.405, E3 +127642.426}
SPL {X  -159.233, Y  +361.951, Z    +0.000, E1   +15.631, E3 +127646.604}
SPL {X  -159.983, Y  +375.952, Z    +0.000, E1    +3.555, E3 +127647.371}
SPL {X  -159.990, Y  +379.545, Z    +0.000, E1    -0.045, E3 +127647.417}
SPL {X  -159.990, Y  +382.058, Z    +0.000, E1    -4.728, E3 +127647.449}
SPL {X  -159.990, Y  +385.965, Z    +0.000, E1   -13.291, E3 +127647.584}
SPL {X  -159.990, Y  +391.054, Z    +0.000, E1   -24.765, E3 +127647.916}
SPL {X  -159.990, Y  +400.233, Z    +0.000, E1   -42.011, E3 +127648.960}
SPL {X  -159.990, Y  +418.500, Z    +0.000, E1   -59.260, E3 +127652.804}
SPL {X  -159.990, Y  +491.183, Z    +0.000, E1   -70.406, E3 +127680.486}
SPL {X  -159.990, Y  +644.105, Z    +0.000, E1   -71.828, E3 +127765.054}
SPL {X  -159.990, Y  +665.410, Z    +0.000, E1   -71.813, E3 +127779.952}
SPL {X  -159.784, Y  +684.619, Z    +0.000, E1   -71.795, E3 +127793.555}
SPL {X  -158.321, Y  +699.551, Z    +0.000, E1   -71.633, E3 +127805.507}
SPL {X  -155.878, Y  +712.540, Z    +0.000, E1   -71.376, E3 +127817.071}
SPL {X  -152.746, Y  +724.097, Z    +0.000, E1   -71.019, E3 +127828.322}
SPL {X  -149.840, Y  +732.578, Z    +0.000, E1   -70.669, E3 +127837.147}
SPL {X  -147.044, Y  +739.548, Z    +0.000, E1   -70.332, E3 +127844.741}
SPL {X  -143.437, Y  +747.371, Z    +0.000, E1   -69.890, E3 +127853.605}
SPL {X  -139.209, Y  +755.353, Z    +0.000, E1   -69.333, E3 +127863.032}
SPL {X  -135.354, Y  +761.800, Z    +0.000, E1   -68.789, E3 +127870.896}
SPL {X  -131.547, Y  +767.562, Z    +0.000, E1   -68.238, E3 +127878.065}
SPL {X  -127.113, Y  +773.655, Z    +0.000, E1   -67.565, E3 +127885.721}
SPL {X  -123.626, Y  +778.056, Z    +0.000, E1   -66.969, E3 +127891.281}
SPL {X   -86.110, Y  +811.340, Z    +0.000, E1   -55.142, E3 +128009.192}
ENDSPLINE

SPLINE
SPL {X  -126.688, Y  +774.208, Z    +0.000, E1   -50.278, E3 +128169.839}
SPL {X  -147.153, Y  +739.291, Z    +0.000, E1   -41.559, E3 +128190.674}
SPL {X  -156.578, Y  +709.366, Z    +0.000, E1   -27.394, E3 +128198.366}
SPL {X  -159.560, Y  +688.227, Z    +0.000, E1   -12.334, E3 +128200.931}
SPL {X  -159.987, Y  +677.470, Z    +0.000, E1    -2.943, E3 +128201.410}
SPL {X  -159.990, Y  +674.465, Z    +0.000, E1    +0.035, E3 +128201.442}
SPL {X  -159.990, Y  +672.210, Z    +0.000, E1    +4.112, E3 +128201.469}
SPL {X  -159.990, Y  +668.446, Z    +0.000, E1   +12.084, E3 +128201.594}
SPL {X  -159.990, Y  +663.424, Z    +0.000, E1   +23.273, E3 +128201.921}
SPL {X  -159.990, Y  +655.288, Z    +0.000, E1   +39.016, E3 +128202.810}
SPL {X  -159.990, Y  +641.020, Z    +0.000, E1   +55.512, E3 +128205.349}
SPL {X  -159.990, Y  +618.237, Z    +0.000, E1   +65.205, E3 +128211.874}
SPL {X  -159.990, Y  +545.807, Z    +0.000, E1   +71.095, E3 +128240.927}
SPL {X  -159.990, Y  +417.971, Z    +0.000, E1   +72.138, E3 +128309.587}
SPL {X  -147.674, Y  +315.943, Z    +0.000, E1   +77.803, E3 +128301.317}
ENDSPLINE

SPLINE
SPL {X  -149.193, Y  +319.722, Z    +0.000, E1   +76.912, E3 +128310.259}
ENDSPLINE

SPLINE
SPL {X  -149.153, Y  +319.620, Z    +0.000, E1   +75.840, E3 +128322.669}
ENDSPLINE

SPLINE
SPL {X  -149.679, Y  +320.993, Z    +0.000, E1   +74.493, E3 +128335.628}
SPL {X  -149.823, Y  +321.377, Z    +0.000, E1   +73.518, E3 +128344.986}
ENDSPLINE

SPLINE
SPL {X  -149.061, Y  +319.382, Z    +0.000, E1   +72.547, E3 +128355.227}
SPL {X  -148.522, Y  +318.020, Z    +0.000, E1   +71.446, E3 +128365.613}
SPL {X  -146.766, Y  +313.809, Z    +0.000, E1   +70.623, E3 +128375.265}
SPL {X  -143.180, Y  +306.112, Z    +0.000, E1   +70.169, E3 +128383.962}
SPL {X  -138.714, Y  +297.780, Z    +0.000, E1   +69.607, E3 +128393.709}
SPL {X  -135.202, Y  +291.959, Z    +0.000, E1   +69.085, E3 +128400.818}
SPL {X  -131.272, Y  +286.043, Z    +0.000, E1   +68.558, E3 +128408.057}
SPL {X  -127.436, Y  +280.769, Z    +0.000, E1   +67.934, E3 +128414.680}
SPL {X  -124.030, Y  +276.439, Z    +0.000, E1   +67.412, E3 +128420.043}
SPL {X   -89.505, Y  +244.889, Z    +0.000, E1   +58.168, E3 +128501.796}
ENDSPLINE

SPLINE
SPL {X  -111.763, Y  +263.019, Z    +0.000, E1   +52.505, E3 +128683.208}
SPL {X  -139.943, Y  +299.958, Z    +0.000, E1   +46.517, E3 +128717.548}
SPL {X  -152.249, Y  +328.336, Z    +0.000, E1   +36.404, E3 +128727.942}
SPL {X  -158.157, Y  +353.354, Z    +0.000, E1   +21.990, E3 +128732.665}
SPL {X  -159.630, Y  +366.769, Z    +0.000, E1   +11.595, E3 +128733.947}
SPL {X  -159.983, Y  +375.952, Z    +0.000, E1    +3.555, E3 +128734.327}
SPL {X  -159.990, Y  +379.545, Z    +0.000, E1    -0.045, E3 +128734.374}
SPL {X  -159.990, Y  +382.058, Z    +0.000, E1    -4.728, E3 +128734.406}
SPL {X  -159.990, Y  +387.492, Z    +0.000, E1   -16.478, E3 +128734.631}
SPL {X  -159.990, Y  +395.172, Z    +0.000, E1   -33.361, E3 +128735.258}
SPL {X  -159.990, Y  +405.626, Z    +0.000, E1   -49.217, E3 +128736.782}
SPL {X  -159.990, Y  +423.679, Z    +0.000, E1   -61.834, E3 +128741.053}
SPL {X  -159.990, Y  +491.183, Z    +0.000, E1   -70.406, E3 +128767.442}
SPL {X  -159.990, Y  +644.105, Z    +0.000, E1   -71.828, E3 +128852.010}
SPL {X  -159.990, Y  +665.410, Z    +0.000, E1   -71.813, E3 +128866.908}
SPL {X  -159.936, Y  +680.656, Z    +0.000, E1   -71.796, E3 +128877.626}
SPL {X  -158.712, Y  +696.685, Z    +0.000, E1   -71.696, E3 +128890.009}
SPL {X  -155.878, Y  +712.540, Z    +0.000, E1   -71.376, E3 +128904.027}
SPL {X  -152.746, Y  +724.097, Z    +0.000, E1   -71.019, E3 +128915.278}
SPL {X  -149.840, Y  +732.578, Z    +0.000, E1   -70.669, E3 +128924.104}
SPL {X  -147.044, Y  +739.548, Z    +0.000, E1   -70.332, E3 +128931.698}
SPL {X  -143.437, Y  +747.371, Z    +0.000, E1   -69.890, E3 +128940.562}
SPL {X  -139.209, Y  +755.353, Z    +0.000, E1   -69.333, E3 +128949.988}
SPL {X  -135.354, Y  +761.800, Z    +0.000, E1   -68.789, E3 +128957.852}
SPL {X  -131.547, Y  +767.562, Z    +0.000, E1   -68.238, E3 +128965.021}
SPL {X  -127.113, Y  +773.655, Z    +0.000, E1   -67.565, E3 +128972.678}
SPL {X  -123.626, Y  +778.056, Z    +0.000, E1   -66.969, E3 +128978.238}
SPL {X   -86.110, Y  +811.340, Z    +0.000, E1   -55.142, E3 +129096.148}
ENDSPLINE

SPLINE
SPL {X  -126.688, Y  +774.208, Z    +0.000, E1   -50.278, E3 +129256.795}
SPL {X  -147.153, Y  +739.291, Z    +0.000, E1   -41.559, E3 +129277.630}
SPL {X  -156.578, Y  +709.366, Z    +0.000, E1   -27.394, E3 +129285.323}
SPL {X  -159.560, Y  +688.227, Z    +0.000, E1   -12.334, E3 +129287.888}
SPL {X  -159.987, Y  +677.470, Z    +0.000, E1    -2.943, E3 +129288.366}
SPL {X  -159.990, Y  +674.465, Z    +0.000, E1    +0.035, E3 +129288.399}
SPL {X  -159.990, Y  +672.210, Z    +0.000, E1    +4.112, E3 +129288.425}
SPL {X  -159.990, Y  +668.446, Z    +0.000, E1   +12.084, E3 +129288.551}
SPL {X  -159.990, Y  +663.424, Z    +0.000, E1   +23.273, E3 +129288.877}
SPL {X  -159.990, Y  +655.288, Z    +0.000, E1   +39.016, E3 +129289.766}
SPL {X  -159.990, Y  +641.020, Z    +0.000, E1   +55.512, E3 +129292.305}
SPL {X  -159.990, Y  +618.237, Z    +0.000, E1   +65.205, E3 +129298.831}
SPL {X  -159.990, Y  +545.807, Z    +0.000, E1   +71.095, E3 +129327.884}
SPL {X  -159.990, Y  +417.971, Z    +0.000, E1   +72.138, E3 +129396.543}
SPL {X  -147.674, Y  +315.943, Z    +0.000, E1   +77.803, E3 +129388.274}
ENDSPLINE

SPLINE
SPL {X  -149.193, Y  +319.722, Z    +0.000, E1   +76.912, E3 +129397.216}
ENDSPLINE

SPLINE
SPL {X  -149.153, Y  +319.620, Z    +0.000, E1   +75.840, E3 +129409.625}
ENDSPLINE

SPLINE
SPL {X  -149.679, Y  +320.993, Z    +0.000, E1   +74.493, E3 +129422.585}
SPL {X  -149.823, Y  +321.377, Z    +0.000, E1   +73.518, E3 +129431.942}
ENDSPLINE

SPLINE
SPL {X  -149.061, Y  +319.382, Z    +0.000, E1   +72.547, E3 +129442.184}
SPL {X  -148.201, Y  +317.223, Z    +0.000, E1   +71.184, E3 +129455.508}
SPL {X  -144.085, Y  +307.957, Z    +0.000, E1   +70.311, E3 +129468.755}
SPL {X  -138.714, Y  +297.780, Z    +0.000, E1   +69.607, E3 +129480.665}
SPL {X  -135.202, Y  +291.959, Z    +0.000, E1   +69.085, E3 +129487.774}
SPL {X  -132.274, Y  +287.498, Z    +0.000, E1   +68.678, E3 +129493.246}
SPL {X  -128.237, Y  +281.834, Z    +0.000, E1   +68.080, E3 +129500.283}
SPL {X  -124.030, Y  +276.439, Z    +0.000, E1   +67.412, E3 +129507.000}
SPL {X   -89.505, Y  +244.889, Z    +0.000, E1   +58.168, E3 +129588.752}
ENDSPLINE

SPLINE
SPL {X  -111.763, Y  +263.019, Z    +0.000, E1   +52.505, E3 +129770.164}
SPL {X  -139.943, Y  +299.958, Z    +0.000, E1   +46.517, E3 +129804.504}
SPL {X  -152.249, Y  +328.336, Z    +0.000, E1   +36.404, E3 +129814.898}
SPL {X  -158.157, Y  +353.354, Z    +0.000, E1   +21.990, E3 +129819.622}
SPL {X  -159.828, Y  +370.311, Z    +0.000, E1    +8.652, E3 +129821.087}
SPL {X  -159.990, Y  +379.415, Z    +0.000, E1    +0.198, E3 +129821.329}
SPL {X  -159.990, Y  +382.058, Z    +0.000, E1    -4.728, E3 +129821.362}
SPL {X  -159.990, Y  +387.492, Z    +0.000, E1   -16.478, E3 +129821.588}
SPL {X  -159.990, Y  +395.172, Z    +0.000, E1   -33.361, E3 +129822.214}
SPL {X  -159.990, Y  +405.626, Z    +0.000, E1   -49.217, E3 +129823.738}
SPL {X  -159.990, Y  +423.679, Z    +0.000, E1   -61.834, E3 +129828.010}
SPL {X  -159.990, Y  +491.183, Z    +0.000, E1   -70.406, E3 +129854.399}
SPL {X  -159.990, Y  +644.105, Z    +0.000, E1   -71.828, E3 +129938.967}
SPL {X  -159.990, Y  +665.410, Z    +0.000, E1   -71.813, E3 +129953.865}
SPL {X  -159.784, Y  +684.619, Z    +0.000, E1   -71.795, E3 +129967.468}
SPL {X  -158.321, Y  +699.551, Z    +0.000, E1   -71.633, E3 +129979.420}
SPL {X  -156.572, Y  +709.392, Z    +0.000, E1   -71.434, E3 +129988.113}
SPL {X  -154.409, Y  +718.389, Z    +0.000, E1   -71.209, E3 +129996.573}
SPL {X  -150.682, Y  +730.275, Z    +0.000, E1   -70.793, E3 +130008.572}
SPL {X  -147.044, Y  +739.548, Z    +0.000, E1   -70.332, E3 +130018.654}
SPL {X  -143.437, Y  +747.371, Z    +0.000, E1   -69.890, E3 +130027.518}
SPL {X  -139.209, Y  +755.353, Z    +0.000, E1   -69.333, E3 +130036.945}
SPL {X  -134.311, Y  +763.433, Z    +0.000, E1   -68.667, E3 +130046.791}
SPL {X  -129.529, Y  +770.410, Z    +0.000, E1   -67.934, E3 +130055.555}
SPL {X  -126.163, Y  +774.886, Z    +0.000, E1   -67.384, E3 +130061.218}
SPL {X  -123.626, Y  +778.056, Z    +0.000, E1   -66.969, E3 +130065.194}
SPL {X   -86.110, Y  +811.340, Z    +0.000, E1   -55.142, E3 +130183.105}
ENDSPLINE

SPLINE
SPL {X  -126.688, Y  +774.208, Z    +0.000, E1   -50.278, E3 +130343.752}
SPL {X  -150.887, Y  +729.697, Z    +0.000, E1   -37.846, E3 +130367.608}
SPL {X  -157.603, Y  +704.031, Z    +0.000, E1   -23.939, E3 +130373.170}
SPL {X  -159.560, Y  +688.227, Z    +0.000, E1   -12.334, E3 +130374.844}
SPL {X  -159.987, Y  +677.470, Z    +0.000, E1    -2.943, E3 +130375.323}
SPL {X  -159.990, Y  +674.465, Z    +0.000, E1    +0.035, E3 +130375.355}
SPL {X  -159.990, Y  +672.210, Z    +0.000, E1    +4.112, E3 +130375.382}
SPL {X  -159.990, Y  +668.446, Z    +0.000, E1   +12.084, E3 +130375.507}
SPL {X  -159.990, Y  +663.424, Z    +0.000, E1   +23.273, E3 +130375.834}
SPL {X  -159.990, Y  +655.288, Z    +0.000, E1   +39.016, E3 +130376.723}
SPL {X  -159.990, Y  +641.020, Z    +0.000, E1   +55.512, E3 +130379.262}
SPL {X  -159.990, Y  +618.237, Z    +0.000, E1   +65.205, E3 +130385.787}
SPL {X  -159.990, Y  +545.807, Z    +0.000, E1   +71.095, E3 +130414.840}
SPL {X  -159.990, Y  +417.971, Z    +0.000, E1   +72.138, E3 +130483.500}
SPL {X  -147.674, Y  +315.943, Z    +0.000, E1   +77.803, E3 +130475.230}
ENDSPLINE

SPLINE
SPL {X  -149.193, Y  +319.722, Z    +0.000, E1   +76.912, E3 +130484.172}
ENDSPLINE

SPLINE
SPL {X  -149.153, Y  +319.620, Z    +0.000, E1   +75.840, E3 +130496.582}
ENDSPLINE

SPLINE
SPL {X  -149.679, Y  +320.993, Z    +0.000, E1   +74.493, E3 +130509.541}
SPL {X  -149.823, Y  +321.377, Z    +0.000, E1   +73.518, E3 +130518.899}
ENDSPLINE

SPLINE
SPL {X  -149.061, Y  +319.382, Z    +0.000, E1   +72.547, E3 +130529.140}
SPL {X  -148.522, Y  +318.020, Z    +0.000, E1   +71.446, E3 +130539.526}
SPL {X  -146.766, Y  +313.809, Z    +0.000, E1   +70.623, E3 +130549.178}
SPL {X  -143.180, Y  +306.112, Z    +0.000, E1   +70.169, E3 +130557.875}
SPL {X  -138.714, Y  +297.780, Z    +0.000, E1   +69.607, E3 +130567.622}
SPL {X  -135.202, Y  +291.959, Z    +0.000, E1   +69.085, E3 +130574.731}
SPL {X  -132.274, Y  +287.498, Z    +0.000, E1   +68.678, E3 +130580.203}
SPL {X  -128.237, Y  +281.834, Z    +0.000, E1   +68.080, E3 +130587.239}
SPL {X  -125.186, Y  +277.874, Z    +0.000, E1   +67.573, E3 +130592.206}
SPL {X  -123.070, Y  +275.272, Z    +0.000, E1   +67.229, E3 +130595.425}
SPL {X   -89.505, Y  +244.889, Z    +0.000, E1   +58.168, E3 +130675.709}
ENDSPLINE

SPLINE
SPL {X  -111.763, Y  +263.019, Z    +0.000, E1   +52.505, E3 +130857.121}
SPL {X  -139.943, Y  +299.958, Z    +0.000, E1   +46.517, E3 +130891.461}
SPL {X  -152.249, Y  +328.336, Z    +0.000, E1   +36.404, E3 +130901.855}
SPL {X  -158.157, Y  +353.354, Z    +0.000, E1   +21.990, E3 +130906.578}
SPL {X  -159.828, Y  +370.311, Z    +0.000, E1    +8.652, E3 +130908.044}
SPL {X  -159.990, Y  +377.723, Z    +0.000, E1    +1.782, E3 +130908.275}
SPL {X  -159.990, Y  +379.545, Z    +0.000, E1    -0.045, E3 +130908.287}
SPL {X  -159.990, Y  +382.058, Z    +0.000, E1    -4.728, E3 +130908.319}
SPL {X  -159.990, Y  +387.492, Z    +0.000, E1   -16.478, E3 +130908.544}
SPL {X  -159.990, Y  +395.172, Z    +0.000, E1   -33.361, E3 +130909.171}
SPL {X  -159.990, Y  +405.626, Z    +0.000, E1   -49.217, E3 +130910.695}
SPL {X  -159.990, Y  +423.679, Z    +0.000, E1   -61.834, E3 +130914.966}
SPL {X  -159.990, Y  +491.183, Z    +0.000, E1   -70.406, E3 +130941.355}
SPL {X  -159.990, Y  +644.105, Z    +0.000, E1   -71.828, E3 +131025.923}
SPL {X  -159.990, Y  +665.410, Z    +0.000, E1   -71.813, E3 +131040.821}
SPL {X  -159.784, Y  +684.619, Z    +0.000, E1   -71.795, E3 +131054.425}
SPL {X  -158.321, Y  +699.551, Z    +0.000, E1   -71.633, E3 +131066.377}
SPL {X  -156.572, Y  +709.392, Z    +0.000, E1   -71.434, E3 +131075.070}
SPL {X  -154.409, Y  +718.389, Z    +0.000, E1   -71.209, E3 +131083.529}
SPL {X  -150.682, Y  +730.275, Z    +0.000, E1   -70.793, E3 +131095.529}
SPL {X  -147.044, Y  +739.548, Z    +0.000, E1   -70.332, E3 +131105.611}
SPL {X  -143.437, Y  +747.371, Z    +0.000, E1   -69.890, E3 +131114.475}
SPL {X  -139.209, Y  +755.353, Z    +0.000, E1   -69.333, E3 +131123.902}
SPL {X  -134.311, Y  +763.433, Z    +0.000, E1   -68.667, E3 +131133.747}
SPL {X  -129.529, Y  +770.410, Z    +0.000, E1   -67.934, E3 +131142.511}
SPL {X  -126.163, Y  +774.886, Z    +0.000, E1   -67.384, E3 +131148.174}
SPL {X  -123.626, Y  +778.056, Z    +0.000, E1   -66.969, E3 +131152.151}
SPL {X   -86.110, Y  +811.340, Z    +0.000, E1   -55.142, E3 +131270.061}
ENDSPLINE

SPLINE
SPL {X  -126.688, Y  +774.208, Z    +0.000, E1   -50.278, E3 +131430.708}
SPL {X  -150.887, Y  +729.697, Z    +0.000, E1   -37.846, E3 +131454.565}
SPL {X  -157.603, Y  +704.031, Z    +0.000, E1   -23.939, E3 +131460.126}
SPL {X  -159.560, Y  +688.227, Z    +0.000, E1   -12.334, E3 +131461.801}
SPL {X  -159.987, Y  +677.470, Z    +0.000, E1    -2.943, E3 +131462.279}
SPL {X  -159.990, Y  +674.465, Z    +0.000, E1    +0.035, E3 +131462.312}
SPL {X  -159.990, Y  +672.210, Z    +0.000, E1    +4.112, E3 +131462.339}
SPL {X  -159.990, Y  +668.446, Z    +0.000, E1   +12.084, E3 +131462.464}
SPL {X  -159.990, Y  +663.424, Z    +0.000, E1   +23.273, E3 +131462.790}
SPL {X  -159.990, Y  +655.288, Z    +0.000, E1   +39.016, E3 +131463.679}
SPL {X  -159.990, Y  +641.020, Z    +0.000, E1   +55.512, E3 +131466.218}
SPL {X  -159.990, Y  +618.237, Z    +0.000, E1   +65.205, E3 +131472.744}
SPL {X  -159.990, Y  +545.807, Z    +0.000, E1   +71.095, E3 +131501.797}
SPL {X  -159.990, Y  +417.971, Z    +0.000, E1   +72.138, E3 +131570.456}
SPL {X  -147.674, Y  +315.943, Z    +0.000, E1   +77.803, E3 +131562.187}
ENDSPLINE

